FUNCTION_BLOCK "LOOP"   // FB2, LAD
{ S7_Optimized_Access := 'TRUE' }
VERSION : 0.1
// stored: AutoNumber true, IsIECCheckEnabled false, IsRetainMemResEnabled false, MemoryReserve 100, SetENOAutomatically false, UDAEnableTagReadback false
   VAR
      PULSO : Bool;
      AuxLoop : Bool;
      N_L00P : Int;
      Aux_N_LOOP : Int;
      Loop : Int;
   END_VAR
   VAR_TEMP   // added for the SCL form of the ladder/FBD networks
      _w1 : Bool;
      _w2 : Bool;
   END_VAR
BEGIN

REGION Network 2
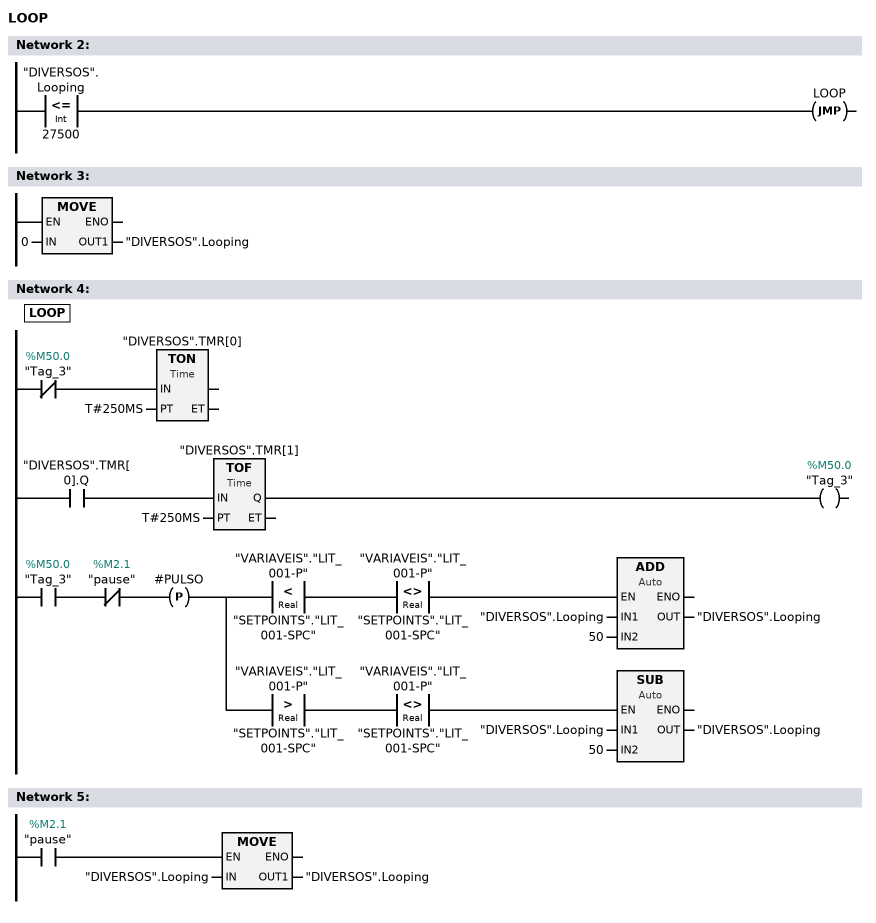
   RUNG wire#powerrail
      { S7_Templates := "SrcType := Int" } LE_Contact(in1 := "DIVERSOS".Looping, in2 := 27500)
      JumpCoil( LOOP )
   END_RUNG
   // the same network as SCL:
   IF "DIVERSOS".Looping <= 27500 THEN GOTO LOOP; END_IF;
END_REGION

REGION Network 3
   RUNG wire#powerrail
      Move(in := 0, out1 => "DIVERSOS".Looping)
   END_RUNG
   // the same network as SCL:
   "DIVERSOS".Looping := 0;
END_REGION

REGION Network 4
   Label( LOOP )
   RUNG wire#powerrail
      I_Contact( "Tag_3" )
      { S7_Templates := "time_type := Time" } "DIVERSOS".TMR[0].TON(pt := T#250MS, et =>)
   END_RUNG
   RUNG wire#powerrail
      Contact( "DIVERSOS".TMR[0].Q )
      { S7_Templates := "time_type := Time" } "DIVERSOS".TMR[1].TOF(pt := T#250MS, et =>)
      Coil( "Tag_3" )
   END_RUNG
   RUNG wire#powerrail
      Contact( "Tag_3" )
      I_Contact( "pause" )
      P_Trig( #PULSO )
      wire#w1
      { S7_Templates := "SrcType := Real" } LT_Contact(in1 := "VARIAVEIS"."LIT_001-P", in2 := "SETPOINTS"."LIT_001-SPC")
      { S7_Templates := "SrcType := Real" } NE_Contact(in1 := "VARIAVEIS"."LIT_001-P", in2 := "SETPOINTS"."LIT_001-SPC")
      Add(in1 := "DIVERSOS".Looping, in2 := 50, out => "DIVERSOS".Looping)
   END_RUNG
   RUNG wire#w1
      { S7_Templates := "SrcType := Real" } GT_Contact(in1 := "VARIAVEIS"."LIT_001-P", in2 := "SETPOINTS"."LIT_001-SPC")
      { S7_Templates := "SrcType := Real" } NE_Contact(in1 := "VARIAVEIS"."LIT_001-P", in2 := "SETPOINTS"."LIT_001-SPC")
      Sub(in1 := "DIVERSOS".Looping, in2 := 50, out => "DIVERSOS".Looping)
   END_RUNG
   // the same network as SCL:
   LOOP:
   "DIVERSOS".TMR[0].TON(IN := NOT "Tag_3", PT := T#250MS);
   "DIVERSOS".TMR[1].TOF(IN := "DIVERSOS".TMR[0].Q, PT := T#250MS);
   "Tag_3" := "DIVERSOS".TMR[1].Q;
   #_w1 := "Tag_3" AND NOT "pause";
   #_w2 := #_w1 AND NOT #PULSO;   // rising edge
   #PULSO := #_w1;
   IF #_w2 AND ("VARIAVEIS"."LIT_001-P" < "SETPOINTS"."LIT_001-SPC") AND ("VARIAVEIS"."LIT_001-P" <> "SETPOINTS"."LIT_001-SPC") THEN
       "DIVERSOS".Looping := "DIVERSOS".Looping + 50;
   END_IF;
   IF #_w2 AND ("VARIAVEIS"."LIT_001-P" > "SETPOINTS"."LIT_001-SPC") AND ("VARIAVEIS"."LIT_001-P" <> "SETPOINTS"."LIT_001-SPC") THEN
       "DIVERSOS".Looping := "DIVERSOS".Looping - 50;
   END_IF;
END_REGION

REGION Network 5
   RUNG wire#powerrail
      Contact( "pause" )
      Move(in := "DIVERSOS".Looping, out1 => "DIVERSOS".Looping)
   END_RUNG
   // the same network as SCL:
   IF "pause" THEN "DIVERSOS".Looping := "DIVERSOS".Looping; END_IF;
END_REGION
END_FUNCTION_BLOCK

FUNCTION_BLOCK "INTPRO"   // FB202, LAD
{ S7_Optimized_Access := 'FALSE' }
VERSION : 0.1
// stored: AutoNumber true, IsIECCheckEnabled false, SetENOAutomatically false, UDAEnableTagReadback false
   VAR DB_SPECIFIC
      EE_P_NIV : Bool;   // HAILITA BOMBA PRINCIPAL PELO NÍVEL
      EE_C1_NIV : Bool;   // HAILITA BOMBA COMPLEMENTAR 1 PELO NÍVEL
      EE_C2_NIV : Bool;   // HAILITA BOMBA COMPLEMENTAR 2 PELO NÍVEL
      EE_P_LS : Bool;   // HAILITA BOMBA PRINCIPAL PELAS BÓIAS
      EE_C1_LS : Bool;   // HAILITA BOMBA COMLEMENTAR 1 PELAS BÓIAS
      EE_C2_LS : Bool;   // HAILITA BOMBA COMPLEMENTAR 2 PELAS BÓIAS
      HAB_P_EE : Bool;   // LIGA BOMBA PRINCIPAL DA ELEVATÓRIA
      HAB_C1_EE : Bool;   // LIGA BOMBA COMPLEMENTAR 1 DA ELEVATÓRIA
      HAB_C2_EE : Bool;   // LIGA BOMBA COMPLEMENTAR 2 DA ELEVATÓRIA
      AUXP01 : Bool;
      BS01OK : Bool;
      BS02OK : Bool;
      BS03OK : Bool;
      L_BS01 : Bool;
      L_BS02 : Bool;
      L_BS03 : Bool;
      AUXP02 : Bool;
      AUXP03 : Bool;
      AUXP04 : Bool;
      AUXP05 : Bool;
      AUXP06 : Bool;
      AUXP07 : Bool;
      ETBS01_T001 : Int;
      ETBS02_T001 : Int;
      ETBS03_T001 : Int;
      BS01TO : Int;
      BS02TO : Int;
      BS03TO : Int;
      BS01TEOK : DInt;
      BS02TEOK : DInt;
      BS03TEOK : DInt;
      TE00 { S7_SetPoint := 'True'} : IEC_TIMER;
   END_VAR
   VAR
      RODEE { S7_SetPoint := 'True'} : "ROD4";
   END_VAR
   VAR_TEMP
      T011S : Int;
      ET_TE00 : Time;
   END_VAR
BEGIN

REGION Network 1: Alarme falha de sinal transmissor de nivel
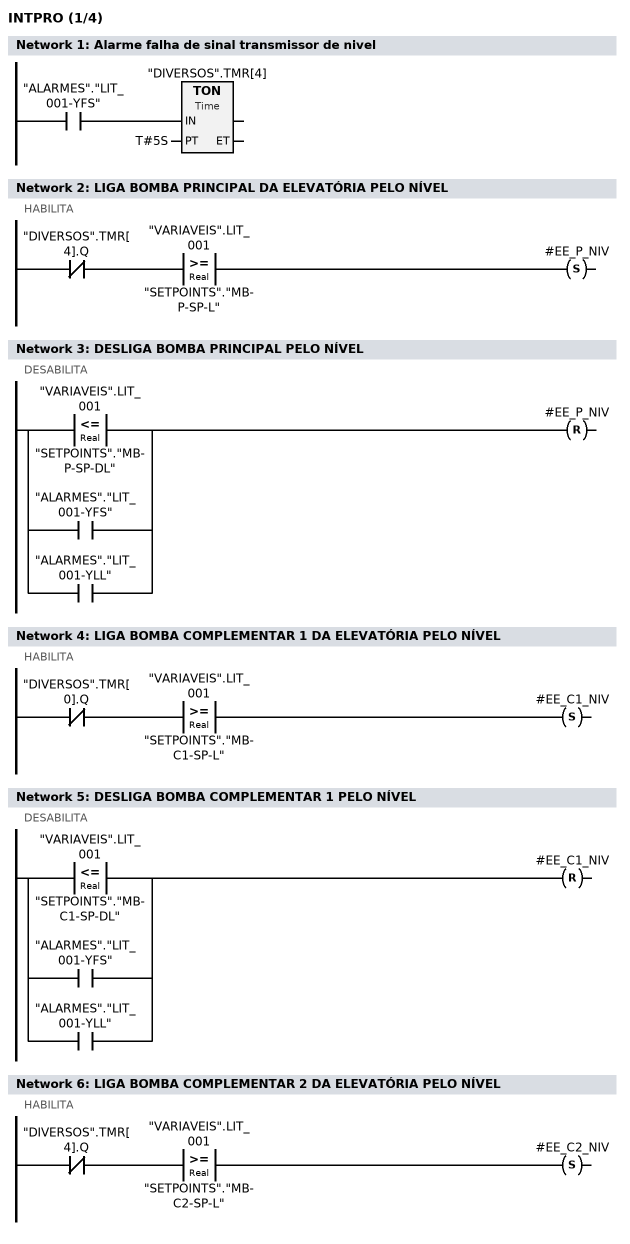
   RUNG wire#powerrail
      Contact( "ALARMES"."LIT_001-YFS" )
      { S7_Templates := "time_type := Time" } "DIVERSOS".TMR[4].TON(pt := T#5S, et =>)
   END_RUNG
   // the same network as SCL:
   "DIVERSOS".TMR[4].TON(IN := "ALARMES"."LIT_001-YFS", PT := T#5S);
END_REGION

REGION Network 2: LIGA BOMBA PRINCIPAL DA ELEVATÓRIA PELO NÍVEL
   // HABILITA
   RUNG wire#powerrail
      I_Contact( "DIVERSOS".TMR[4].Q )
      { S7_Templates := "SrcType := Real" } GE_Contact(in1 := "VARIAVEIS".LIT_001, in2 := "SETPOINTS"."MB-P-SP-L")
      S_Coil( #EE_P_NIV )
   END_RUNG
   // the same network as SCL:
   IF NOT "DIVERSOS".TMR[4].Q AND ("VARIAVEIS".LIT_001 >= "SETPOINTS"."MB-P-SP-L") THEN
       #EE_P_NIV := TRUE;
   END_IF;
END_REGION

REGION Network 3: DESLIGA BOMBA PRINCIPAL PELO NÍVEL
   // DESABILITA
   RUNG wire#powerrail
      { S7_Templates := "SrcType := Real" } LE_Contact(in1 := "VARIAVEIS".LIT_001, in2 := "SETPOINTS"."MB-P-SP-DL")
      wire#w1
      R_Coil( #EE_P_NIV )
   END_RUNG
   RUNG wire#powerrail
      Contact( "ALARMES"."LIT_001-YFS" )
   END_RUNG wire#w1
   RUNG wire#powerrail
      Contact( "ALARMES"."LIT_001-YLL" )
   END_RUNG wire#w1
   // the same network as SCL:
   IF ("VARIAVEIS".LIT_001 <= "SETPOINTS"."MB-P-SP-DL") OR "ALARMES"."LIT_001-YFS" OR "ALARMES"."LIT_001-YLL" THEN
       #EE_P_NIV := FALSE;
   END_IF;
END_REGION

REGION Network 4: LIGA BOMBA COMPLEMENTAR 1 DA ELEVATÓRIA PELO NÍVEL
   // HABILITA
   RUNG wire#powerrail
      I_Contact( "DIVERSOS".TMR[0].Q )
      { S7_Templates := "SrcType := Real" } GE_Contact(in1 := "VARIAVEIS".LIT_001, in2 := "SETPOINTS"."MB-C1-SP-L")
      S_Coil( #EE_C1_NIV )
   END_RUNG
   // the same network as SCL:
   IF NOT "DIVERSOS".TMR[0].Q AND ("VARIAVEIS".LIT_001 >= "SETPOINTS"."MB-C1-SP-L") THEN
       #EE_C1_NIV := TRUE;
   END_IF;
END_REGION

REGION Network 5: DESLIGA BOMBA COMPLEMENTAR 1 PELO NÍVEL
   // DESABILITA
   RUNG wire#powerrail
      { S7_Templates := "SrcType := Real" } LE_Contact(in1 := "VARIAVEIS".LIT_001, in2 := "SETPOINTS"."MB-C1-SP-DL")
      wire#w1
      R_Coil( #EE_C1_NIV )
   END_RUNG
   RUNG wire#powerrail
      Contact( "ALARMES"."LIT_001-YFS" )
   END_RUNG wire#w1
   RUNG wire#powerrail
      Contact( "ALARMES"."LIT_001-YLL" )
   END_RUNG wire#w1
   // the same network as SCL:
   IF ("VARIAVEIS".LIT_001 <= "SETPOINTS"."MB-C1-SP-DL") OR "ALARMES"."LIT_001-YFS" OR "ALARMES"."LIT_001-YLL" THEN
       #EE_C1_NIV := FALSE;
   END_IF;
END_REGION

REGION Network 6: LIGA BOMBA COMPLEMENTAR 2 DA ELEVATÓRIA PELO NÍVEL
   // HABILITA
   RUNG wire#powerrail
      I_Contact( "DIVERSOS".TMR[4].Q )
      { S7_Templates := "SrcType := Real" } GE_Contact(in1 := "VARIAVEIS".LIT_001, in2 := "SETPOINTS"."MB-C2-SP-L")
      S_Coil( #EE_C2_NIV )
   END_RUNG
   // the same network as SCL:
   IF NOT "DIVERSOS".TMR[4].Q AND ("VARIAVEIS".LIT_001 >= "SETPOINTS"."MB-C2-SP-L") THEN
       #EE_C2_NIV := TRUE;
   END_IF;
END_REGION

REGION Network 7: DESLIGA BOMBA COMPLEMENTAR 2 PELO NÍVEL
   // DESABILITA
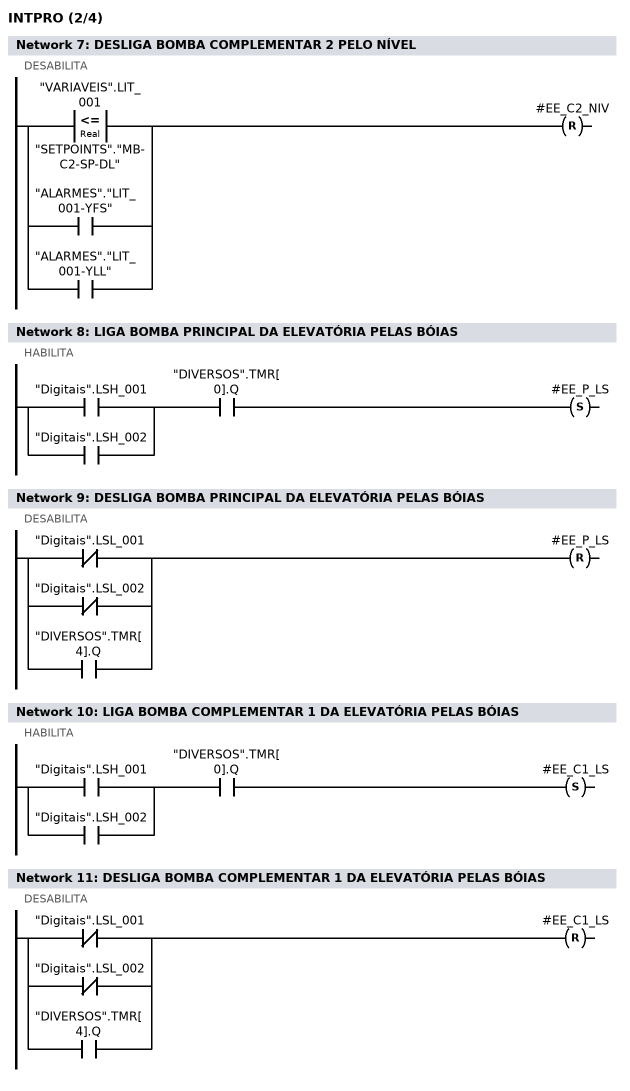
   RUNG wire#powerrail
      { S7_Templates := "SrcType := Real" } LE_Contact(in1 := "VARIAVEIS".LIT_001, in2 := "SETPOINTS"."MB-C2-SP-DL")
      wire#w1
      R_Coil( #EE_C2_NIV )
   END_RUNG
   RUNG wire#powerrail
      Contact( "ALARMES"."LIT_001-YFS" )
   END_RUNG wire#w1
   RUNG wire#powerrail
      Contact( "ALARMES"."LIT_001-YLL" )
   END_RUNG wire#w1
   // the same network as SCL:
   IF ("VARIAVEIS".LIT_001 <= "SETPOINTS"."MB-C2-SP-DL") OR "ALARMES"."LIT_001-YFS" OR "ALARMES"."LIT_001-YLL" THEN
       #EE_C2_NIV := FALSE;
   END_IF;
END_REGION

REGION Network 8: LIGA BOMBA PRINCIPAL DA ELEVATÓRIA PELAS BÓIAS
   // HABILITA
   RUNG wire#powerrail
      Contact( "Digitais".LSH_001 )
      wire#w1
      Contact( "DIVERSOS".TMR[0].Q )
      S_Coil( #EE_P_LS )
   END_RUNG
   RUNG wire#powerrail
      Contact( "Digitais".LSH_002 )
   END_RUNG wire#w1
   // the same network as SCL:
   IF ("Digitais".LSH_001 OR "Digitais".LSH_002) AND "DIVERSOS".TMR[0].Q THEN #EE_P_LS := TRUE; END_IF;
END_REGION

REGION Network 9: DESLIGA BOMBA PRINCIPAL DA ELEVATÓRIA PELAS BÓIAS
   // DESABILITA
   RUNG wire#powerrail
      I_Contact( "Digitais".LSL_001 )
      wire#w1
      R_Coil( #EE_P_LS )
   END_RUNG
   RUNG wire#powerrail
      I_Contact( "Digitais".LSL_002 )
   END_RUNG wire#w1
   RUNG wire#powerrail
      Contact( "DIVERSOS".TMR[4].Q )
   END_RUNG wire#w1
   // the same network as SCL:
   IF NOT "Digitais".LSL_001 OR NOT "Digitais".LSL_002 OR "DIVERSOS".TMR[4].Q THEN #EE_P_LS := FALSE; END_IF;
END_REGION

REGION Network 10: LIGA BOMBA COMPLEMENTAR 1 DA ELEVATÓRIA PELAS BÓIAS
   // HABILITA
   RUNG wire#powerrail
      Contact( "Digitais".LSH_001 )
      wire#w1
      Contact( "DIVERSOS".TMR[0].Q )
      S_Coil( #EE_C1_LS )
   END_RUNG
   RUNG wire#powerrail
      Contact( "Digitais".LSH_002 )
   END_RUNG wire#w1
   // the same network as SCL:
   IF ("Digitais".LSH_001 OR "Digitais".LSH_002) AND "DIVERSOS".TMR[0].Q THEN #EE_C1_LS := TRUE; END_IF;
END_REGION

REGION Network 11: DESLIGA BOMBA COMPLEMENTAR 1 DA ELEVATÓRIA PELAS BÓIAS
   // DESABILITA
   RUNG wire#powerrail
      I_Contact( "Digitais".LSL_001 )
      wire#w1
      R_Coil( #EE_C1_LS )
   END_RUNG
   RUNG wire#powerrail
      I_Contact( "Digitais".LSL_002 )
   END_RUNG wire#w1
   RUNG wire#powerrail
      Contact( "DIVERSOS".TMR[4].Q )
   END_RUNG wire#w1
   // the same network as SCL:
   IF NOT "Digitais".LSL_001 OR NOT "Digitais".LSL_002 OR "DIVERSOS".TMR[4].Q THEN
       #EE_C1_LS := FALSE;
   END_IF;
END_REGION

REGION Network 12: LIGA BOMBA COMPLEMENTAR 2 DA ELEVATÓRIA PELAS BÓIAS
   // HABILITA
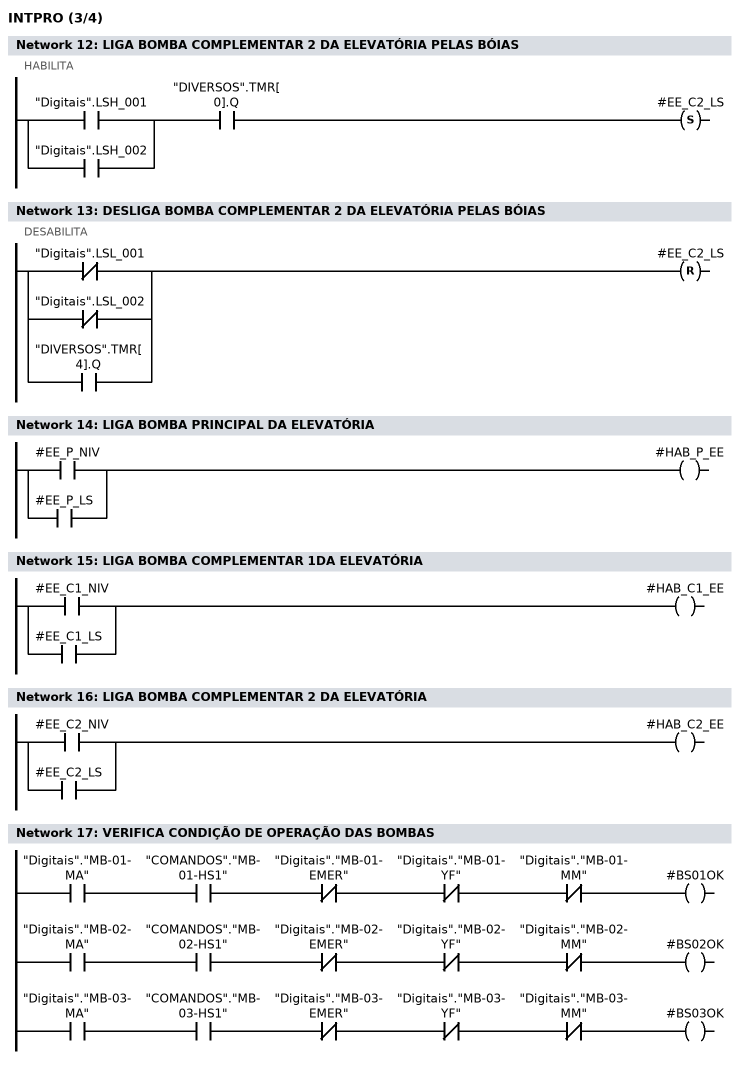
   RUNG wire#powerrail
      Contact( "Digitais".LSH_001 )
      wire#w1
      Contact( "DIVERSOS".TMR[0].Q )
      S_Coil( #EE_C2_LS )
   END_RUNG
   RUNG wire#powerrail
      Contact( "Digitais".LSH_002 )
   END_RUNG wire#w1
   // the same network as SCL:
   IF ("Digitais".LSH_001 OR "Digitais".LSH_002) AND "DIVERSOS".TMR[0].Q THEN #EE_C2_LS := TRUE; END_IF;
END_REGION

REGION Network 13: DESLIGA BOMBA COMPLEMENTAR 2 DA ELEVATÓRIA PELAS BÓIAS
   // DESABILITA
   RUNG wire#powerrail
      I_Contact( "Digitais".LSL_001 )
      wire#w1
      R_Coil( #EE_C2_LS )
   END_RUNG
   RUNG wire#powerrail
      I_Contact( "Digitais".LSL_002 )
   END_RUNG wire#w1
   RUNG wire#powerrail
      Contact( "DIVERSOS".TMR[4].Q )
   END_RUNG wire#w1
   // the same network as SCL:
   IF NOT "Digitais".LSL_001 OR NOT "Digitais".LSL_002 OR "DIVERSOS".TMR[4].Q THEN
       #EE_C2_LS := FALSE;
   END_IF;
END_REGION

REGION Network 14: LIGA BOMBA PRINCIPAL DA ELEVATÓRIA
   RUNG wire#powerrail
      Contact( #EE_P_NIV )
      wire#w1
      Coil( #HAB_P_EE )
   END_RUNG
   RUNG wire#powerrail
      Contact( #EE_P_LS )
   END_RUNG wire#w1
   // the same network as SCL:
   #HAB_P_EE := #EE_P_NIV OR #EE_P_LS;
END_REGION

REGION Network 15: LIGA BOMBA COMPLEMENTAR 1DA ELEVATÓRIA
   RUNG wire#powerrail
      Contact( #EE_C1_NIV )
      wire#w1
      Coil( #HAB_C1_EE )
   END_RUNG
   RUNG wire#powerrail
      Contact( #EE_C1_LS )
   END_RUNG wire#w1
   // the same network as SCL:
   #HAB_C1_EE := #EE_C1_NIV OR #EE_C1_LS;
END_REGION

REGION Network 16: LIGA BOMBA COMPLEMENTAR 2 DA ELEVATÓRIA
   RUNG wire#powerrail
      Contact( #EE_C2_NIV )
      wire#w1
      Coil( #HAB_C2_EE )
   END_RUNG
   RUNG wire#powerrail
      Contact( #EE_C2_LS )
   END_RUNG wire#w1
   // the same network as SCL:
   #HAB_C2_EE := #EE_C2_NIV OR #EE_C2_LS;
END_REGION

REGION Network 17: VERIFICA CONDIÇÃO DE OPERAÇÃO DAS BOMBAS
   RUNG wire#powerrail
      Contact( "Digitais"."MB-01-MA" )
      Contact( "COMANDOS"."MB-01-HS1" )
      I_Contact( "Digitais"."MB-01-EMER" )
      I_Contact( "Digitais"."MB-01-YF" )
      I_Contact( "Digitais"."MB-01-MM" )
      Coil( #BS01OK )
   END_RUNG
   RUNG wire#powerrail
      Contact( "Digitais"."MB-02-MA" )
      Contact( "COMANDOS"."MB-02-HS1" )
      I_Contact( "Digitais"."MB-02-EMER" )
      I_Contact( "Digitais"."MB-02-YF" )
      I_Contact( "Digitais"."MB-02-MM" )
      Coil( #BS02OK )
   END_RUNG
   RUNG wire#powerrail
      Contact( "Digitais"."MB-03-MA" )
      Contact( "COMANDOS"."MB-03-HS1" )
      I_Contact( "Digitais"."MB-03-EMER" )
      I_Contact( "Digitais"."MB-03-YF" )
      I_Contact( "Digitais"."MB-03-MM" )
      Coil( #BS03OK )
   END_RUNG
   // the same network as SCL:
   #BS01OK := "Digitais"."MB-01-MA" AND "COMANDOS"."MB-01-HS1" AND NOT "Digitais"."MB-01-EMER" AND NOT "Digitais"."MB-01-YF" AND NOT "Digitais"."MB-01-MM";
   #BS02OK := "Digitais"."MB-02-MA" AND "COMANDOS"."MB-02-HS1" AND NOT "Digitais"."MB-02-EMER" AND NOT "Digitais"."MB-02-YF" AND NOT "Digitais"."MB-02-MM";
   #BS03OK := "Digitais"."MB-03-MA" AND "COMANDOS"."MB-03-HS1" AND NOT "Digitais"."MB-03-EMER" AND NOT "Digitais"."MB-03-YF" AND NOT "Digitais"."MB-03-MM";
END_REGION

REGION Network 18: RODÍZIO DAS BOMBAS
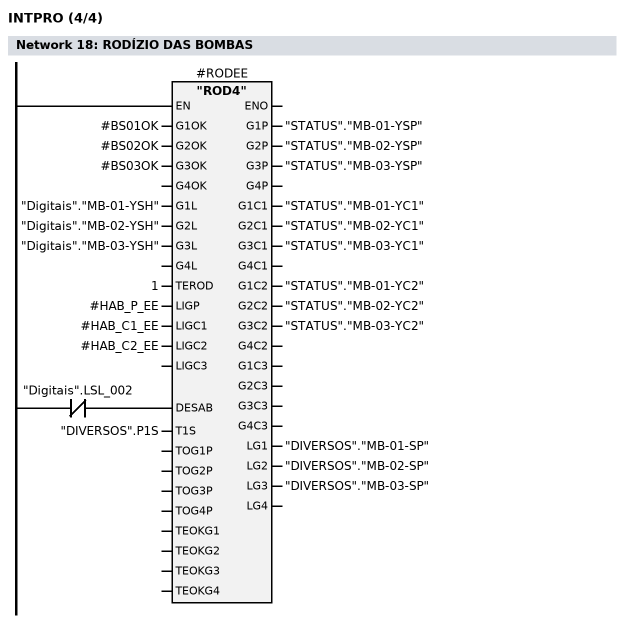
   RUNG wire#powerrail
      #RODEE(DESAB := wire#w1, G1OK := #BS01OK, G2OK := #BS02OK, G3OK := #BS03OK, G4OK :=, G1L := "Digitais"."MB-01-YSH", G2L := "Digitais"."MB-02-YSH", G3L := "Digitais"."MB-03-YSH", G4L :=, TEROD := 1, LIGP := #HAB_P_EE, LIGC1 := #HAB_C1_EE, LIGC2 := #HAB_C2_EE, LIGC3 :=, T1S := "DIVERSOS".P1S, TOG1P :=, TOG2P :=, TOG3P :=, TOG4P :=, TEOKG1 :=, TEOKG2 :=, TEOKG3 :=, TEOKG4 :=, G1P => "STATUS"."MB-01-YSP", G2P => "STATUS"."MB-02-YSP", G3P => "STATUS"."MB-03-YSP", G4P =>, G1C1 => "STATUS"."MB-01-YC1", G2C1 => "STATUS"."MB-02-YC1", G3C1 => "STATUS"."MB-03-YC1", G4C1 =>, G1C2 => "STATUS"."MB-01-YC2", G2C2 => "STATUS"."MB-02-YC2", G3C2 => "STATUS"."MB-03-YC2", G4C2 =>, G1C3 =>, G2C3 =>, G3C3 =>, G4C3 =>, LG1 => "DIVERSOS"."MB-01-SP", LG2 => "DIVERSOS"."MB-02-SP", LG3 => "DIVERSOS"."MB-03-SP", LG4 =>)
   END_RUNG
   RUNG wire#powerrail
      I_Contact( "Digitais".LSL_002 )
   END_RUNG wire#w1
   // the same network as SCL:
   #RODEE(G1OK := #BS01OK,   // "ROD4"
          G2OK := #BS02OK,
          G3OK := #BS03OK,
          G1L := "Digitais"."MB-01-YSH",
          G2L := "Digitais"."MB-02-YSH",
          G3L := "Digitais"."MB-03-YSH",
          TEROD := 1,
          LIGP := #HAB_P_EE,
          LIGC1 := #HAB_C1_EE,
          LIGC2 := #HAB_C2_EE,
          DESAB := NOT "Digitais".LSL_002,
          T1S := "DIVERSOS".P1S,
          G1P => "STATUS"."MB-01-YSP",
          G2P => "STATUS"."MB-02-YSP",
          G3P => "STATUS"."MB-03-YSP",
          G1C1 => "STATUS"."MB-01-YC1",
          G2C1 => "STATUS"."MB-02-YC1",
          G3C1 => "STATUS"."MB-03-YC1",
          G1C2 => "STATUS"."MB-01-YC2",
          G2C2 => "STATUS"."MB-02-YC2",
          G3C2 => "STATUS"."MB-03-YC2",
          LG1 => "DIVERSOS"."MB-01-SP",
          LG2 => "DIVERSOS"."MB-02-SP",
          LG3 => "DIVERSOS"."MB-03-SP");
END_REGION
END_FUNCTION_BLOCK

FUNCTION_BLOCK "ROD4"   // FB200, LAD
TITLE = Rodízio de 4 grupos
{ S7_Optimized_Access := 'FALSE' }
VERSION : 0.1
// stored: AutoNumber false, IsIECCheckEnabled false, SetENOAutomatically false, UDAEnableTagReadback false
   VAR_INPUT
      G1OK : Bool;   // GRUPO EM CONDIÇÕES DE OPERAÇÃO
      G2OK : Bool;   // GRUPO EM CONDIÇÕES DE OPERAÇÃO
      G3OK : Bool;   // GRUPO EM CONDIÇÕES DE OPERAÇÃO
      G4OK : Bool;   // GRUPO EM CONDIÇÕES DE OPERAÇÃO
      G1L : Bool;   // GRUPO LIGADO
      G2L : Bool;   // GRUPO LIGADO
      G3L : Bool;   // GRUPO LIGADO
      G4L : Bool;   // GRUPO LIGADO
      TEROD : DInt;   // TEMPOPARA RODÍZIO DAS BOMBAS
      LIGP : Bool;   // LIGA BOMBA PRINCIPAL
      LIGC1 : Bool;   // LIGA BOMBA COMPLEMENTAR 1
      LIGC2 : Bool;   // LIGA BOMBA COMPLEMENTAR 2
      LIGC3 : Bool;   // LIGA BOMBA COMPLEMENTAR 3
      DESAB : Bool;   // DESABILITA FUNCIONAMENTO DOS GRUPOS
      T1S : Bool;   // PULSO A CADA 1 SEGUNDO
   END_VAR
   VAR_OUTPUT
      G1P : Bool;   // GRUPO 1 SELECIONADO COMO PRINCIPAL
      G2P : Bool;   // GRUPO 2 SELECIONADO COMO PRINCIPAL
      G3P : Bool;   // GRUPO 3 SELECIONADO COMO PRINCIPAL
      G4P : Bool;   // GRUPO 4 SELECIONADO COMO PRINCIPAL
      G1C1 : Bool;   // GRUPO 1 SELECIONADO COMO COMPLEMENTAR 1
      G2C1 : Bool;   // GRUPO 2 SELECIONADO COMO COMPLEMENTAR 1
      G3C1 : Bool;   // GRUPO 3 SELECIONADO COMO COMPLEMENTAR 1
      G4C1 : Bool;   // GRUPO 4 SELECIONADO COMO COMPLEMENTAR 1
      G1C2 : Bool;   // GRUPO 1 SELECIONADO COMO COMPLEMENTAR 2
      G2C2 : Bool;   // GRUPO 2 SELECIONADO COMO COMPLEMENTAR 2
      G3C2 : Bool;   // GRUPO 3 SELECIONADO COMO COMPLEMENTAR 3
      G4C2 : Bool;   // GRUPO 4 SELECIONADO COMO COMPLEMENTAR 4
      G1C3 : Bool;   // GRUPO 1 SELECIONADO COMO COMPLEMENTAR 3
      G2C3 : Bool;   // GRUPO 2 SELECIONADO COMO COMPLEMENTAR 3
      G3C3 : Bool;   // GRUPO 3 SELECIONADO COMO COMPLEMENTAR 3
      G4C3 : Bool;   // GRUPO 4 SELECIONADO COMO COMPLEMENTAR 3
      LG1 : Bool;   // LIGA GRUPO 1
      LG2 : Bool;   // LIGA GRUPO 2
      LG3 : Bool;   // LIGA GRUPO 3
      LG4 : Bool;   // LIGA GRUPO 4
   END_VAR
   VAR_IN_OUT
      TOG1P : DInt;   // TEMPO DE OPERAÇÃO GRUPO 1
      TOG2P : DInt;   // TEMPO DE OPERAÇÃO GRUPO 2
      TOG3P : DInt;   // TEMPO DE OPERAÇÃO GRUPO 3
      TOG4P : DInt;   // TEMPO DE OPERAÇÃO GRUPO 4
      TEOKG1 : Real;   // TEMPO OK GRUPO 1
      TEOKG2 : Real;   // TEMPO OK GRUPO 2
      TEOKG3 : Real;   // TEMPO OK GRUPO 3
      TEOKG4 : Real;   // TEMPO OK GRUPO 4
   END_VAR
   VAR DB_SPECIFIC
      GR1SELP : Bool;   // SELECIONADO COMO PRINCIPAL
      GR2SELP : Bool;   // SELECIONADO COMO PRINCIPAL
      GR3SELP : Bool;   // SELECIONADO COMO PRINCIPAL
      GR4SELP : Bool;   // SELECIONADO COMO PRINCIPAL
      GR1SELC1 : Bool;   // SELECIONADO COMO COMPLEMENTAR 1
      GR2SELC1 : Bool;   // SELECIONADO COMO COMPLEMENTAR 1
      GR3SELC1 : Bool;   // SELECIONADO COMO COMPLEMENTAR 1
      GR4SELC1 : Bool;   // SELECIONADO COMO COMPLEMENTAR 1
      GR1SELC2 : Bool;   // SELECIONADO COMO COMPLEMENTAR 2
      GR2SELC2 : Bool;   // SELECIONADO COMO COMPLEMENTAR 2
      GR3SELC2 : Bool;   // SELECIONADO COMO COMPLEMENTAR 2
      GR4SELC2 : Bool;   // SELECIONADO COMO COMPLEMENTAR 2
      GR1SELC3 : Bool;   // SELECIONADO COMO COMPLEMENTAR 3
      GR2SELC3 : Bool;   // SELECIONADO COMO COMPLEMENTAR 3
      GR3SELC3 : Bool;   // SELECIONADO COMO COMPLEMENTAR 3
      GR4SELC3 : Bool;   // SELECIONADO COMO COMPLEMENTAR 3
      PS1SG1 : Bool;   // AUXILIAR DE PULSO
      PS1SG2 : Bool;   // AUXILIAR DE PULSO
      PS1SG3 : Bool;   // AUXILIAR DE PULSO
      PS1SG4 : Bool;   // AUXILIAR DE PULSO
      PS1 : Bool;   // AUXILIAR DE PULSO
      PS2 : Bool;   // AUXILIAR DE PULSO
      PS3 : Bool;   // AUXILIAR DE PULSO
      PS4 : Bool;   // AUXILIAR DE PULSO
      FIMTEG1 : Bool;   // FIM DO TEMPO DE EXISTÊNCIA DO GRUPO 1
      FIMTEG2 : Bool;   // FIM DO TEMPO DE EXISTÊNCIA DO GRUPO 2
      FIMTEG3 : Bool;   // FIM DO TEMPO DE EXISTÊNCIA DO GRUPO 3
      FIMTEG4 : Bool;   // FIM DO TEMPO DE EXISTÊNCIA DO GRUPO 4
      SDESG1 : Bool;   // SOLICITAÇÃO DE DESLIGAMENTO
      SDESG2 : Bool;   // SOLICITAÇÃO DE DESLIGAMENTO
      SDESG3 : Bool;   // SOLICITAÇÃO DE DESLIGAMENTO
      SDESG4 : Bool;   // SOLICITAÇÃO DE DESLIGAMENTO
      GPL : Bool;   // GRUPO PRINCIPAL LIGADO
      GC1L : Bool;   // GRUPO COMPLEMENTAR 1 LIGADO
      GC2L : Bool;   // GRUPO COMPLEMENTAR 2 LIGADO
      GC3L : Bool;   // GRUPO COMPLEMENTAR 3 LIGADO
      SO_L : Bool;   // SOLICITAÇÃO DE PARTIDA
      SO_D : Bool;   // SOLICITAÇÃO DE DESLIGAMENTO
      RTEOKG1 : Bool;   // RESET TEMPO OK
      RTEOKG2 : Bool;   // RESET TEMPO OK
      RTEOKG3 : Bool;   // RESET TEMPO OK
      RTEOKG4 : Bool;   // RESET TEMPO OK
      TON1 { S7_SetPoint := 'True'} : TON_TIME;   // TEMPORIZADOR
      TON2 { S7_SetPoint := 'True'} : TON_TIME;   // TEMPORIZADOR
      TON3 { S7_SetPoint := 'True'} : TON_TIME;   // TEMPORIZADOR
      TON4 { S7_SetPoint := 'True'} : TON_TIME;   // TEMPORIZADOR
      TSDG1 { S7_SetPoint := 'True'} : TON_TIME;   // TEMPORIZADOR
      TSDG2 { S7_SetPoint := 'True'} : TON_TIME;   // TEMPORIZADOR
      TSDG3 { S7_SetPoint := 'True'} : TON_TIME;   // TEMPORIZADOR
      TSDG4 { S7_SetPoint := 'True'} : TON_TIME;   // TEMPORIZADOR
   END_VAR
   VAR_TEMP
      PRI12 : Bool;   // PRIORIDADE GRUPO 1
      PRI13 : Bool;   // PRIORIDADE GRUPO 1
      PRI14 : Bool;   // PRIORIDADE GRUPO 1
      PRI23 : Bool;   // PRIORIDADE GRUPO 2
      PRI24 : Bool;   // PRIORIDADE GRUPO 2
      PRI34 : Bool;   // PRIORIDADE GRUPO 3
      TMROD : Real;   // TEMPO DE RODIZIO
      NGS : Int;   // NÚMERO DE GRUPOS SOLICITADOS
      NGF : Int;   // NÚMERO DE GRUPOS FUNCIONANDO
      AUX01 : Int;   // AUXILIAR UTILIZADO NA LÓGICA
      AUX02 : Int;   // AUXILIAR UTILIZADO NA LÓGICA
      AUX03 : Int;   // AUXILIAR UTILIZADO NA LÓGICA
      AUX04 : Int;   // AUXILIAR UTILIZADO NA LÓGICA
      AUX05 : Bool;   // AUXILIAR UTILIZADO NA LÓGICA
      AUX06 : Bool;   // AUXILIAR UTILIZADO NA LÓGICA
      AUX07 : Bool;   // AUXILIAR UTILIZADO NA LÓGICA
      AUX08 : Bool;   // AUXILIAR UTILIZADO NA LÓGICA
      ETT1 : Time;   // EFETIVO DO TEMPORIZADOR
      ETT2 : Time;   // EFETIVO DO TEMPORIZADOR
      ETT3 : Time;   // EFETIVO DO TEMPORIZADOR
      ETT4 : Time;   // EFETIVO DO TEMPORIZADOR
      ETTSDG4 : Time;   // EFETIVO DO TEMPORIZADOR
      ETTSDG3 : Time;   // EFETIVO DO TEMPORIZADOR
      ETTSDG2 : Time;   // EFETIVO DO TEMPORIZADOR
      ETTSDG1 : Time;   // EFETIVO DO TEMPORIZADOR
   END_VAR
   VAR_TEMP   // added for the SCL form of the ladder/FBD networks
      _w1 : Bool;
   END_VAR
BEGIN

REGION Network 1: Tranforme em segundo o tempo de rodízio dos sopradores
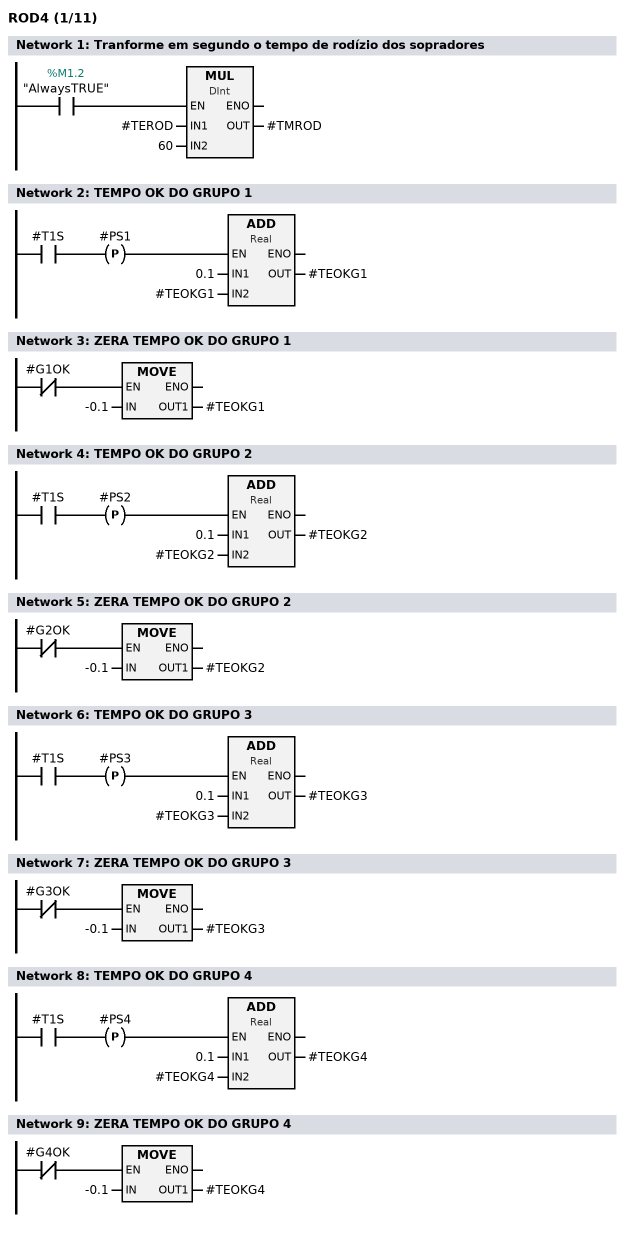
   RUNG wire#powerrail
      Contact( "AlwaysTRUE" )
      { S7_Templates := "SrcType := DInt"; S7_GenerateENO := "TRUE" } Mul(in1 := #TEROD, in2 := 60, out => #TMROD)
   END_RUNG
   // the same network as SCL:
   IF "AlwaysTRUE" THEN #TMROD := #TEROD * 60; END_IF;
END_REGION

REGION Network 2: TEMPO OK DO GRUPO 1
   RUNG wire#powerrail
      Contact( #T1S )
      P_Trig( #PS1 )
      { S7_Templates := "SrcType := Real"; S7_GenerateENO := "TRUE" } Add(in1 := 0.1, in2 := #TEOKG1, out => #TEOKG1)
   END_RUNG
   // the same network as SCL:
   #_w1 := #T1S AND NOT #PS1;   // rising edge
   #PS1 := #T1S;
   IF #_w1 THEN #TEOKG1 := 0.1 + #TEOKG1; END_IF;
END_REGION

REGION Network 3: ZERA TEMPO OK DO GRUPO 1
   RUNG wire#powerrail
      I_Contact( #G1OK )
      { S7_GenerateENO := "TRUE" } Move(in := -0.1, out1 => #TEOKG1)
   END_RUNG
   // the same network as SCL:
   IF NOT #G1OK THEN #TEOKG1 := -0.1; END_IF;
END_REGION

REGION Network 4: TEMPO OK DO GRUPO 2
   RUNG wire#powerrail
      Contact( #T1S )
      P_Trig( #PS2 )
      { S7_Templates := "SrcType := Real"; S7_GenerateENO := "TRUE" } Add(in1 := 0.1, in2 := #TEOKG2, out => #TEOKG2)
   END_RUNG
   // the same network as SCL:
   #_w1 := #T1S AND NOT #PS2;   // rising edge
   #PS2 := #T1S;
   IF #_w1 THEN #TEOKG2 := 0.1 + #TEOKG2; END_IF;
END_REGION

REGION Network 5: ZERA TEMPO OK DO GRUPO 2
   RUNG wire#powerrail
      I_Contact( #G2OK )
      { S7_GenerateENO := "TRUE" } Move(in := -0.1, out1 => #TEOKG2)
   END_RUNG
   // the same network as SCL:
   IF NOT #G2OK THEN #TEOKG2 := -0.1; END_IF;
END_REGION

REGION Network 6: TEMPO OK DO GRUPO 3
   RUNG wire#powerrail
      Contact( #T1S )
      P_Trig( #PS3 )
      { S7_Templates := "SrcType := Real"; S7_GenerateENO := "TRUE" } Add(in1 := 0.1, in2 := #TEOKG3, out => #TEOKG3)
   END_RUNG
   // the same network as SCL:
   #_w1 := #T1S AND NOT #PS3;   // rising edge
   #PS3 := #T1S;
   IF #_w1 THEN #TEOKG3 := 0.1 + #TEOKG3; END_IF;
END_REGION

REGION Network 7: ZERA TEMPO OK DO GRUPO 3
   RUNG wire#powerrail
      I_Contact( #G3OK )
      { S7_GenerateENO := "TRUE" } Move(in := -0.1, out1 => #TEOKG3)
   END_RUNG
   // the same network as SCL:
   IF NOT #G3OK THEN #TEOKG3 := -0.1; END_IF;
END_REGION

REGION Network 8: TEMPO OK DO GRUPO 4
   RUNG wire#powerrail
      Contact( #T1S )
      P_Trig( #PS4 )
      { S7_Templates := "SrcType := Real"; S7_GenerateENO := "TRUE" } Add(in1 := 0.1, in2 := #TEOKG4, out => #TEOKG4)
   END_RUNG
   // the same network as SCL:
   #_w1 := #T1S AND NOT #PS4;   // rising edge
   #PS4 := #T1S;
   IF #_w1 THEN #TEOKG4 := 0.1 + #TEOKG4; END_IF;
END_REGION

REGION Network 9: ZERA TEMPO OK DO GRUPO 4
   RUNG wire#powerrail
      I_Contact( #G4OK )
      { S7_GenerateENO := "TRUE" } Move(in := -0.1, out1 => #TEOKG4)
   END_RUNG
   // the same network as SCL:
   IF NOT #G4OK THEN #TEOKG4 := -0.1; END_IF;
END_REGION

REGION Network 10: DEFINIÇÇÃO DE PRIORIDADE DO GRUPO 1
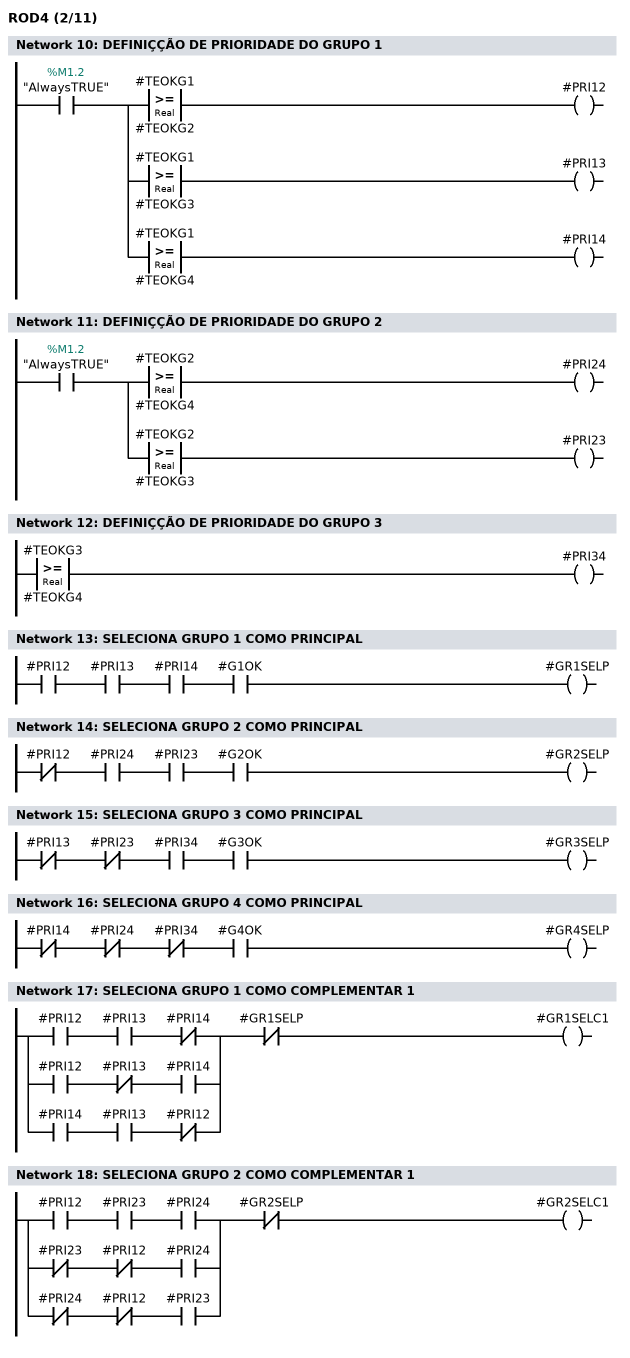
   RUNG wire#powerrail
      Contact( "AlwaysTRUE" )
      wire#w1
      { S7_Templates := "SrcType := Real" } GE_Contact(in1 := #TEOKG1, in2 := #TEOKG2)
      Coil( #PRI12 )
   END_RUNG
   RUNG wire#w1
      { S7_Templates := "SrcType := Real" } GE_Contact(in1 := #TEOKG1, in2 := #TEOKG3)
      Coil( #PRI13 )
   END_RUNG
   RUNG wire#w1
      { S7_Templates := "SrcType := Real" } GE_Contact(in1 := #TEOKG1, in2 := #TEOKG4)
      Coil( #PRI14 )
   END_RUNG
   // the same network as SCL:
   #PRI12 := "AlwaysTRUE" AND (#TEOKG1 >= #TEOKG2);
   #PRI13 := "AlwaysTRUE" AND (#TEOKG1 >= #TEOKG3);
   #PRI14 := "AlwaysTRUE" AND (#TEOKG1 >= #TEOKG4);
END_REGION

REGION Network 11: DEFINIÇÇÃO DE PRIORIDADE DO GRUPO 2
   RUNG wire#powerrail
      Contact( "AlwaysTRUE" )
      wire#w1
      { S7_Templates := "SrcType := Real" } GE_Contact(in1 := #TEOKG2, in2 := #TEOKG4)
      Coil( #PRI24 )
   END_RUNG
   RUNG wire#w1
      { S7_Templates := "SrcType := Real" } GE_Contact(in1 := #TEOKG2, in2 := #TEOKG3)
      Coil( #PRI23 )
   END_RUNG
   // the same network as SCL:
   #PRI24 := "AlwaysTRUE" AND (#TEOKG2 >= #TEOKG4);
   #PRI23 := "AlwaysTRUE" AND (#TEOKG2 >= #TEOKG3);
END_REGION

REGION Network 12: DEFINIÇÇÃO DE PRIORIDADE DO GRUPO 3
   RUNG wire#powerrail
      { S7_Templates := "SrcType := Real" } GE_Contact(in1 := #TEOKG3, in2 := #TEOKG4)
      Coil( #PRI34 )
   END_RUNG
   // the same network as SCL:
   #PRI34 := #TEOKG3 >= #TEOKG4;
END_REGION

REGION Network 13: SELECIONA GRUPO 1 COMO PRINCIPAL
   RUNG wire#powerrail
      Contact( #PRI12 )
      Contact( #PRI13 )
      Contact( #PRI14 )
      Contact( #G1OK )
      Coil( #GR1SELP )
   END_RUNG
   // the same network as SCL:
   #GR1SELP := #PRI12 AND #PRI13 AND #PRI14 AND #G1OK;
END_REGION

REGION Network 14: SELECIONA GRUPO 2 COMO PRINCIPAL
   RUNG wire#powerrail
      I_Contact( #PRI12 )
      Contact( #PRI24 )
      Contact( #PRI23 )
      Contact( #G2OK )
      Coil( #GR2SELP )
   END_RUNG
   // the same network as SCL:
   #GR2SELP := NOT #PRI12 AND #PRI24 AND #PRI23 AND #G2OK;
END_REGION

REGION Network 15: SELECIONA GRUPO 3 COMO PRINCIPAL
   RUNG wire#powerrail
      I_Contact( #PRI13 )
      I_Contact( #PRI23 )
      Contact( #PRI34 )
      Contact( #G3OK )
      Coil( #GR3SELP )
   END_RUNG
   // the same network as SCL:
   #GR3SELP := NOT #PRI13 AND NOT #PRI23 AND #PRI34 AND #G3OK;
END_REGION

REGION Network 16: SELECIONA GRUPO 4 COMO PRINCIPAL
   RUNG wire#powerrail
      I_Contact( #PRI14 )
      I_Contact( #PRI24 )
      I_Contact( #PRI34 )
      Contact( #G4OK )
      Coil( #GR4SELP )
   END_RUNG
   // the same network as SCL:
   #GR4SELP := NOT #PRI14 AND NOT #PRI24 AND NOT #PRI34 AND #G4OK;
END_REGION

REGION Network 17: SELECIONA GRUPO 1 COMO COMPLEMENTAR 1
   RUNG wire#powerrail
      Contact( #PRI12 )
      Contact( #PRI13 )
      I_Contact( #PRI14 )
      wire#w1
      I_Contact( #GR1SELP )
      Coil( #GR1SELC1 )
   END_RUNG
   RUNG wire#powerrail
      Contact( #PRI12 )
      I_Contact( #PRI13 )
      Contact( #PRI14 )
   END_RUNG wire#w1
   RUNG wire#powerrail
      Contact( #PRI14 )
      Contact( #PRI13 )
      I_Contact( #PRI12 )
   END_RUNG wire#w1
   // the same network as SCL:
   #GR1SELC1 := ((#PRI12 AND #PRI13 AND NOT #PRI14) OR (#PRI12 AND NOT #PRI13 AND #PRI14) OR (#PRI14 AND #PRI13 AND NOT #PRI12)) AND NOT #GR1SELP;
END_REGION

REGION Network 18: SELECIONA GRUPO 2 COMO COMPLEMENTAR 1
   RUNG wire#powerrail
      Contact( #PRI12 )
      Contact( #PRI23 )
      Contact( #PRI24 )
      wire#w1
      I_Contact( #GR2SELP )
      Coil( #GR2SELC1 )
   END_RUNG
   RUNG wire#powerrail
      I_Contact( #PRI23 )
      I_Contact( #PRI12 )
      Contact( #PRI24 )
   END_RUNG wire#w1
   RUNG wire#powerrail
      I_Contact( #PRI24 )
      I_Contact( #PRI12 )
      Contact( #PRI23 )
   END_RUNG wire#w1
   // the same network as SCL:
   #GR2SELC1 := ((#PRI12 AND #PRI23 AND #PRI24) OR (NOT #PRI23 AND NOT #PRI12 AND #PRI24) OR (NOT #PRI24 AND NOT #PRI12 AND #PRI23)) AND NOT #GR2SELP;
END_REGION

REGION Network 19: SELECIONA GRUPO 3 COMO COMPLEMENTAR 1
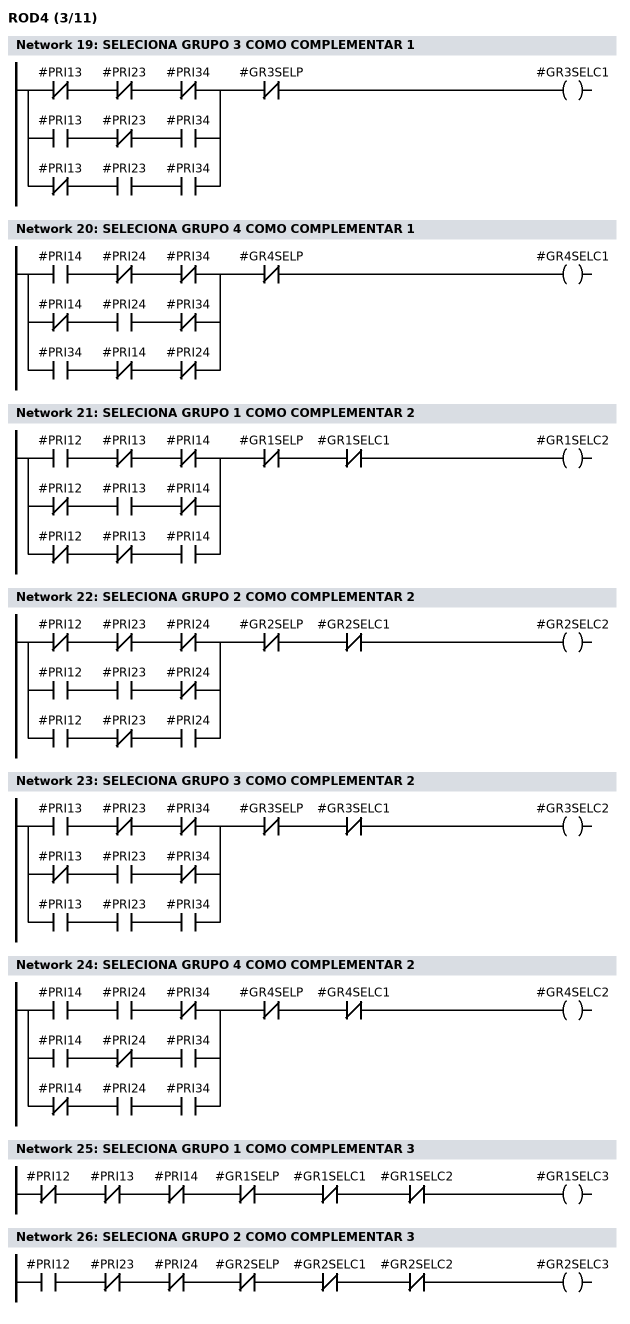
   RUNG wire#powerrail
      I_Contact( #PRI13 )
      I_Contact( #PRI23 )
      I_Contact( #PRI34 )
      wire#w1
      I_Contact( #GR3SELP )
      Coil( #GR3SELC1 )
   END_RUNG
   RUNG wire#powerrail
      Contact( #PRI13 )
      I_Contact( #PRI23 )
      Contact( #PRI34 )
   END_RUNG wire#w1
   RUNG wire#powerrail
      I_Contact( #PRI13 )
      Contact( #PRI23 )
      Contact( #PRI34 )
   END_RUNG wire#w1
   // the same network as SCL:
   #GR3SELC1 := ((NOT #PRI13 AND NOT #PRI23 AND NOT #PRI34) OR (#PRI13 AND NOT #PRI23 AND #PRI34) OR (NOT #PRI13 AND #PRI23 AND #PRI34)) AND NOT #GR3SELP;
END_REGION

REGION Network 20: SELECIONA GRUPO 4 COMO COMPLEMENTAR 1
   RUNG wire#powerrail
      Contact( #PRI14 )
      I_Contact( #PRI24 )
      I_Contact( #PRI34 )
      wire#w1
      I_Contact( #GR4SELP )
      Coil( #GR4SELC1 )
   END_RUNG
   RUNG wire#powerrail
      I_Contact( #PRI14 )
      Contact( #PRI24 )
      I_Contact( #PRI34 )
   END_RUNG wire#w1
   RUNG wire#powerrail
      Contact( #PRI34 )
      I_Contact( #PRI14 )
      I_Contact( #PRI24 )
   END_RUNG wire#w1
   // the same network as SCL:
   #GR4SELC1 := ((#PRI14 AND NOT #PRI24 AND NOT #PRI34) OR (NOT #PRI14 AND #PRI24 AND NOT #PRI34) OR (#PRI34 AND NOT #PRI14 AND NOT #PRI24)) AND NOT #GR4SELP;
END_REGION

REGION Network 21: SELECIONA GRUPO 1 COMO COMPLEMENTAR 2
   RUNG wire#powerrail
      Contact( #PRI12 )
      I_Contact( #PRI13 )
      I_Contact( #PRI14 )
      wire#w1
      I_Contact( #GR1SELP )
      I_Contact( #GR1SELC1 )
      Coil( #GR1SELC2 )
   END_RUNG
   RUNG wire#powerrail
      I_Contact( #PRI12 )
      Contact( #PRI13 )
      I_Contact( #PRI14 )
   END_RUNG wire#w1
   RUNG wire#powerrail
      I_Contact( #PRI12 )
      I_Contact( #PRI13 )
      Contact( #PRI14 )
   END_RUNG wire#w1
   // the same network as SCL:
   #GR1SELC2 := ((#PRI12 AND NOT #PRI13 AND NOT #PRI14) OR (NOT #PRI12 AND #PRI13 AND NOT #PRI14) OR (NOT #PRI12 AND NOT #PRI13 AND #PRI14)) AND NOT #GR1SELP AND NOT #GR1SELC1;
END_REGION

REGION Network 22: SELECIONA GRUPO 2 COMO COMPLEMENTAR 2
   RUNG wire#powerrail
      I_Contact( #PRI12 )
      I_Contact( #PRI23 )
      I_Contact( #PRI24 )
      wire#w1
      I_Contact( #GR2SELP )
      I_Contact( #GR2SELC1 )
      Coil( #GR2SELC2 )
   END_RUNG
   RUNG wire#powerrail
      Contact( #PRI12 )
      Contact( #PRI23 )
      I_Contact( #PRI24 )
   END_RUNG wire#w1
   RUNG wire#powerrail
      Contact( #PRI12 )
      I_Contact( #PRI23 )
      Contact( #PRI24 )
   END_RUNG wire#w1
   // the same network as SCL:
   #GR2SELC2 := ((NOT #PRI12 AND NOT #PRI23 AND NOT #PRI24) OR (#PRI12 AND #PRI23 AND NOT #PRI24) OR (#PRI12 AND NOT #PRI23 AND #PRI24)) AND NOT #GR2SELP AND NOT #GR2SELC1;
END_REGION

REGION Network 23: SELECIONA GRUPO 3 COMO COMPLEMENTAR 2
   RUNG wire#powerrail
      Contact( #PRI13 )
      I_Contact( #PRI23 )
      I_Contact( #PRI34 )
      wire#w1
      I_Contact( #GR3SELP )
      I_Contact( #GR3SELC1 )
      Coil( #GR3SELC2 )
   END_RUNG
   RUNG wire#powerrail
      I_Contact( #PRI13 )
      Contact( #PRI23 )
      I_Contact( #PRI34 )
   END_RUNG wire#w1
   RUNG wire#powerrail
      Contact( #PRI13 )
      Contact( #PRI23 )
      Contact( #PRI34 )
   END_RUNG wire#w1
   // the same network as SCL:
   #GR3SELC2 := ((#PRI13 AND NOT #PRI23 AND NOT #PRI34) OR (NOT #PRI13 AND #PRI23 AND NOT #PRI34) OR (#PRI13 AND #PRI23 AND #PRI34)) AND NOT #GR3SELP AND NOT #GR3SELC1;
END_REGION

REGION Network 24: SELECIONA GRUPO 4 COMO COMPLEMENTAR 2
   RUNG wire#powerrail
      Contact( #PRI14 )
      Contact( #PRI24 )
      I_Contact( #PRI34 )
      wire#w1
      I_Contact( #GR4SELP )
      I_Contact( #GR4SELC1 )
      Coil( #GR4SELC2 )
   END_RUNG
   RUNG wire#powerrail
      Contact( #PRI14 )
      I_Contact( #PRI24 )
      Contact( #PRI34 )
   END_RUNG wire#w1
   RUNG wire#powerrail
      I_Contact( #PRI14 )
      Contact( #PRI24 )
      Contact( #PRI34 )
   END_RUNG wire#w1
   // the same network as SCL:
   #GR4SELC2 := ((#PRI14 AND #PRI24 AND NOT #PRI34) OR (#PRI14 AND NOT #PRI24 AND #PRI34) OR (NOT #PRI14 AND #PRI24 AND #PRI34)) AND NOT #GR4SELP AND NOT #GR4SELC1;
END_REGION

REGION Network 25: SELECIONA GRUPO 1 COMO COMPLEMENTAR 3
   RUNG wire#powerrail
      I_Contact( #PRI12 )
      I_Contact( #PRI13 )
      I_Contact( #PRI14 )
      I_Contact( #GR1SELP )
      I_Contact( #GR1SELC1 )
      I_Contact( #GR1SELC2 )
      Coil( #GR1SELC3 )
   END_RUNG
   // the same network as SCL:
   #GR1SELC3 := NOT #PRI12 AND NOT #PRI13 AND NOT #PRI14 AND NOT #GR1SELP AND NOT #GR1SELC1 AND NOT #GR1SELC2;
END_REGION

REGION Network 26: SELECIONA GRUPO 2 COMO COMPLEMENTAR 3
   RUNG wire#powerrail
      Contact( #PRI12 )
      I_Contact( #PRI23 )
      I_Contact( #PRI24 )
      I_Contact( #GR2SELP )
      I_Contact( #GR2SELC1 )
      I_Contact( #GR2SELC2 )
      Coil( #GR2SELC3 )
   END_RUNG
   // the same network as SCL:
   #GR2SELC3 := #PRI12 AND NOT #PRI23 AND NOT #PRI24 AND NOT #GR2SELP AND NOT #GR2SELC1 AND NOT #GR2SELC2;
END_REGION

REGION Network 27: SELECIONA GRUPO 3 COMO COMPLEMENTAR 3
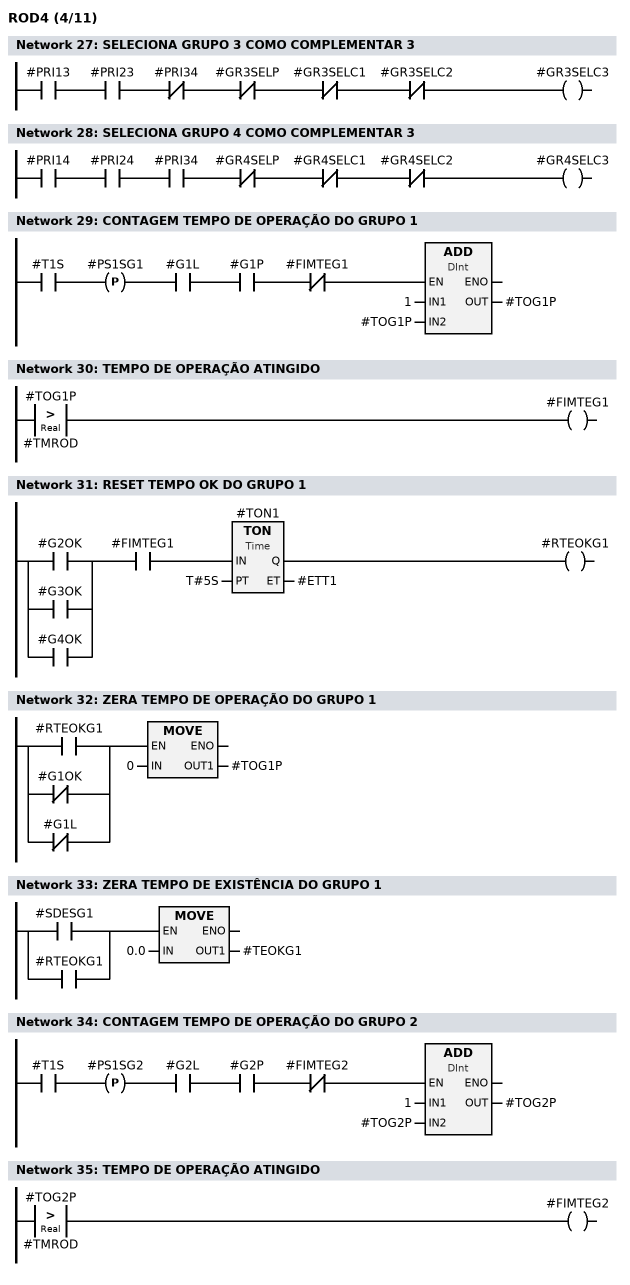
   RUNG wire#powerrail
      Contact( #PRI13 )
      Contact( #PRI23 )
      I_Contact( #PRI34 )
      I_Contact( #GR3SELP )
      I_Contact( #GR3SELC1 )
      I_Contact( #GR3SELC2 )
      Coil( #GR3SELC3 )
   END_RUNG
   // the same network as SCL:
   #GR3SELC3 := #PRI13 AND #PRI23 AND NOT #PRI34 AND NOT #GR3SELP AND NOT #GR3SELC1 AND NOT #GR3SELC2;
END_REGION

REGION Network 28: SELECIONA GRUPO 4 COMO COMPLEMENTAR 3
   RUNG wire#powerrail
      Contact( #PRI14 )
      Contact( #PRI24 )
      Contact( #PRI34 )
      I_Contact( #GR4SELP )
      I_Contact( #GR4SELC1 )
      I_Contact( #GR4SELC2 )
      Coil( #GR4SELC3 )
   END_RUNG
   // the same network as SCL:
   #GR4SELC3 := #PRI14 AND #PRI24 AND #PRI34 AND NOT #GR4SELP AND NOT #GR4SELC1 AND NOT #GR4SELC2;
END_REGION

REGION Network 29: CONTAGEM TEMPO DE OPERAÇÃO DO GRUPO 1
   RUNG wire#powerrail
      Contact( #T1S )
      P_Trig( #PS1SG1 )
      Contact( #G1L )
      Contact( #G1P )
      I_Contact( #FIMTEG1 )
      { S7_Templates := "SrcType := DInt"; S7_GenerateENO := "TRUE" } Add(in1 := 1, in2 := #TOG1P, out => #TOG1P)
   END_RUNG
   // the same network as SCL:
   #_w1 := #T1S AND NOT #PS1SG1;   // rising edge
   #PS1SG1 := #T1S;
   IF #_w1 AND #G1L AND #G1P AND NOT #FIMTEG1 THEN #TOG1P := 1 + #TOG1P; END_IF;
END_REGION

REGION Network 30: TEMPO DE OPERAÇÃO ATINGIDO
   RUNG wire#powerrail
      { S7_Templates := "SrcType := Real" } GT_Contact(in1 := #TOG1P, in2 := #TMROD)
      Coil( #FIMTEG1 )
   END_RUNG
   // the same network as SCL:
   #FIMTEG1 := #TOG1P > #TMROD;
END_REGION

REGION Network 31: RESET TEMPO OK DO GRUPO 1
   RUNG wire#powerrail
      Contact( #G2OK )
      wire#w1
      Contact( #FIMTEG1 )
      { S7_Templates := "time_type := Time" } #TON1.TON(pt := T#5S, et => #ETT1)
      Coil( #RTEOKG1 )
   END_RUNG
   RUNG wire#powerrail
      Contact( #G3OK )
   END_RUNG wire#w1
   RUNG wire#powerrail
      Contact( #G4OK )
   END_RUNG wire#w1
   // the same network as SCL:
   #TON1(IN := (#G2OK OR #G3OK OR #G4OK) AND #FIMTEG1, PT := T#5S, ET => #ETT1);   // TON
   #RTEOKG1 := #TON1.Q;
END_REGION

REGION Network 32: ZERA TEMPO DE OPERAÇÃO DO GRUPO 1
   RUNG wire#powerrail
      Contact( #RTEOKG1 )
      wire#w1
      { S7_GenerateENO := "TRUE" } Move(in := 0, out1 => #TOG1P)
   END_RUNG
   RUNG wire#powerrail
      I_Contact( #G1OK )
   END_RUNG wire#w1
   RUNG wire#powerrail
      I_Contact( #G1L )
   END_RUNG wire#w1
   // the same network as SCL:
   IF #RTEOKG1 OR NOT #G1OK OR NOT #G1L THEN #TOG1P := 0; END_IF;
END_REGION

REGION Network 33: ZERA TEMPO DE EXISTÊNCIA DO GRUPO 1
   RUNG wire#powerrail
      Contact( #SDESG1 )
      wire#w1
      { S7_GenerateENO := "TRUE" } Move(in := 0.0, out1 => #TEOKG1)
   END_RUNG
   RUNG wire#powerrail
      Contact( #RTEOKG1 )
   END_RUNG wire#w1
   // the same network as SCL:
   IF #SDESG1 OR #RTEOKG1 THEN #TEOKG1 := 0.0; END_IF;
END_REGION

REGION Network 34: CONTAGEM TEMPO DE OPERAÇÃO DO GRUPO 2
   RUNG wire#powerrail
      Contact( #T1S )
      P_Trig( #PS1SG2 )
      Contact( #G2L )
      Contact( #G2P )
      I_Contact( #FIMTEG2 )
      { S7_Templates := "SrcType := DInt"; S7_GenerateENO := "TRUE" } Add(in1 := 1, in2 := #TOG2P, out => #TOG2P)
   END_RUNG
   // the same network as SCL:
   #_w1 := #T1S AND NOT #PS1SG2;   // rising edge
   #PS1SG2 := #T1S;
   IF #_w1 AND #G2L AND #G2P AND NOT #FIMTEG2 THEN #TOG2P := 1 + #TOG2P; END_IF;
END_REGION

REGION Network 35: TEMPO DE OPERAÇÃO ATINGIDO
   RUNG wire#powerrail
      { S7_Templates := "SrcType := Real" } GT_Contact(in1 := #TOG2P, in2 := #TMROD)
      Coil( #FIMTEG2 )
   END_RUNG
   // the same network as SCL:
   #FIMTEG2 := #TOG2P > #TMROD;
END_REGION

REGION Network 36: RESET TEMPO OK DO GRUPO 2
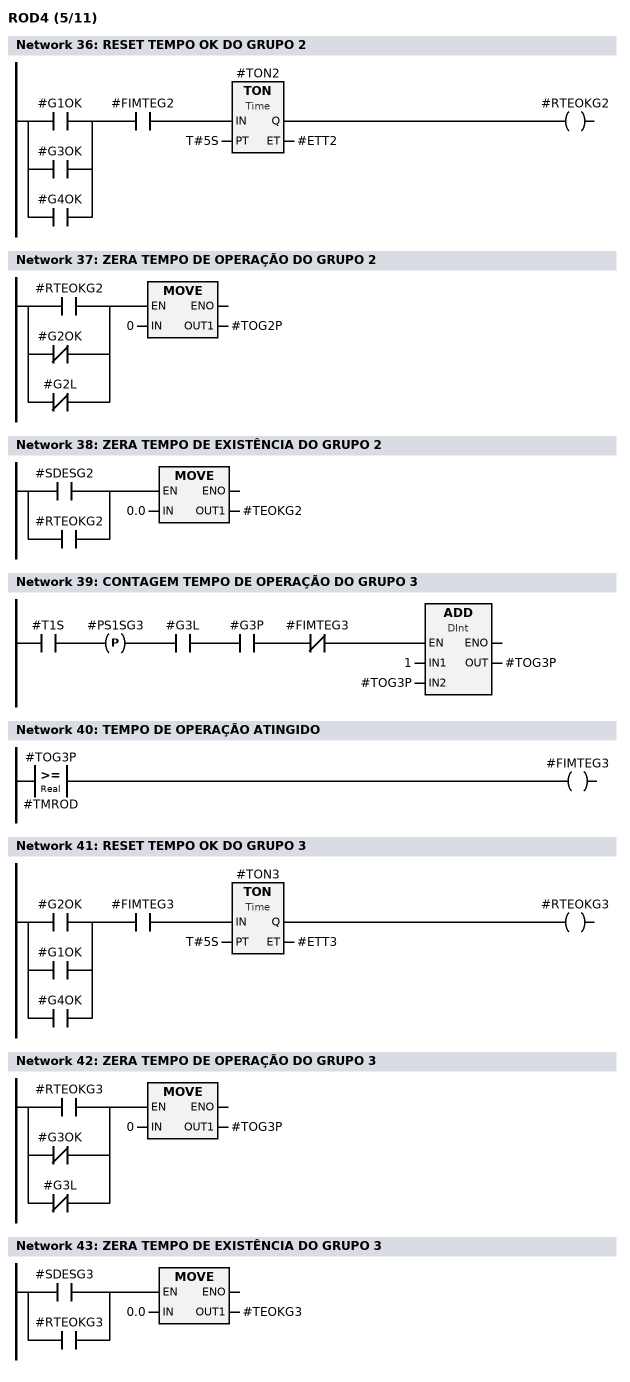
   RUNG wire#powerrail
      Contact( #G1OK )
      wire#w1
      Contact( #FIMTEG2 )
      { S7_Templates := "time_type := Time" } #TON2.TON(pt := T#5S, et => #ETT2)
      Coil( #RTEOKG2 )
   END_RUNG
   RUNG wire#powerrail
      Contact( #G3OK )
   END_RUNG wire#w1
   RUNG wire#powerrail
      Contact( #G4OK )
   END_RUNG wire#w1
   // the same network as SCL:
   #TON2(IN := (#G1OK OR #G3OK OR #G4OK) AND #FIMTEG2, PT := T#5S, ET => #ETT2);   // TON
   #RTEOKG2 := #TON2.Q;
END_REGION

REGION Network 37: ZERA TEMPO DE OPERAÇÃO DO GRUPO 2
   RUNG wire#powerrail
      Contact( #RTEOKG2 )
      wire#w1
      { S7_GenerateENO := "TRUE" } Move(in := 0, out1 => #TOG2P)
   END_RUNG
   RUNG wire#powerrail
      I_Contact( #G2OK )
   END_RUNG wire#w1
   RUNG wire#powerrail
      I_Contact( #G2L )
   END_RUNG wire#w1
   // the same network as SCL:
   IF #RTEOKG2 OR NOT #G2OK OR NOT #G2L THEN #TOG2P := 0; END_IF;
END_REGION

REGION Network 38: ZERA TEMPO DE EXISTÊNCIA DO GRUPO 2
   RUNG wire#powerrail
      Contact( #SDESG2 )
      wire#w1
      { S7_GenerateENO := "TRUE" } Move(in := 0.0, out1 => #TEOKG2)
   END_RUNG
   RUNG wire#powerrail
      Contact( #RTEOKG2 )
   END_RUNG wire#w1
   // the same network as SCL:
   IF #SDESG2 OR #RTEOKG2 THEN #TEOKG2 := 0.0; END_IF;
END_REGION

REGION Network 39: CONTAGEM TEMPO DE OPERAÇÃO DO GRUPO 3
   RUNG wire#powerrail
      Contact( #T1S )
      P_Trig( #PS1SG3 )
      Contact( #G3L )
      Contact( #G3P )
      I_Contact( #FIMTEG3 )
      { S7_Templates := "SrcType := DInt"; S7_GenerateENO := "TRUE" } Add(in1 := 1, in2 := #TOG3P, out => #TOG3P)
   END_RUNG
   // the same network as SCL:
   #_w1 := #T1S AND NOT #PS1SG3;   // rising edge
   #PS1SG3 := #T1S;
   IF #_w1 AND #G3L AND #G3P AND NOT #FIMTEG3 THEN #TOG3P := 1 + #TOG3P; END_IF;
END_REGION

REGION Network 40: TEMPO DE OPERAÇÃO ATINGIDO
   RUNG wire#powerrail
      { S7_Templates := "SrcType := Real" } GE_Contact(in1 := #TOG3P, in2 := #TMROD)
      Coil( #FIMTEG3 )
   END_RUNG
   // the same network as SCL:
   #FIMTEG3 := #TOG3P >= #TMROD;
END_REGION

REGION Network 41: RESET TEMPO OK DO GRUPO 3
   RUNG wire#powerrail
      Contact( #G2OK )
      wire#w1
      Contact( #FIMTEG3 )
      { S7_Templates := "time_type := Time" } #TON3.TON(pt := T#5S, et => #ETT3)
      Coil( #RTEOKG3 )
   END_RUNG
   RUNG wire#powerrail
      Contact( #G1OK )
   END_RUNG wire#w1
   RUNG wire#powerrail
      Contact( #G4OK )
   END_RUNG wire#w1
   // the same network as SCL:
   #TON3(IN := (#G2OK OR #G1OK OR #G4OK) AND #FIMTEG3, PT := T#5S, ET => #ETT3);   // TON
   #RTEOKG3 := #TON3.Q;
END_REGION

REGION Network 42: ZERA TEMPO DE OPERAÇÃO DO GRUPO 3
   RUNG wire#powerrail
      Contact( #RTEOKG3 )
      wire#w1
      { S7_GenerateENO := "TRUE" } Move(in := 0, out1 => #TOG3P)
   END_RUNG
   RUNG wire#powerrail
      I_Contact( #G3OK )
   END_RUNG wire#w1
   RUNG wire#powerrail
      I_Contact( #G3L )
   END_RUNG wire#w1
   // the same network as SCL:
   IF #RTEOKG3 OR NOT #G3OK OR NOT #G3L THEN #TOG3P := 0; END_IF;
END_REGION

REGION Network 43: ZERA TEMPO DE EXISTÊNCIA DO GRUPO 3
   RUNG wire#powerrail
      Contact( #SDESG3 )
      wire#w1
      { S7_GenerateENO := "TRUE" } Move(in := 0.0, out1 => #TEOKG3)
   END_RUNG
   RUNG wire#powerrail
      Contact( #RTEOKG3 )
   END_RUNG wire#w1
   // the same network as SCL:
   IF #SDESG3 OR #RTEOKG3 THEN #TEOKG3 := 0.0; END_IF;
END_REGION

REGION Network 44: CONTAGEM TEMPO DE OPERAÇÃO DO GRUPO 4
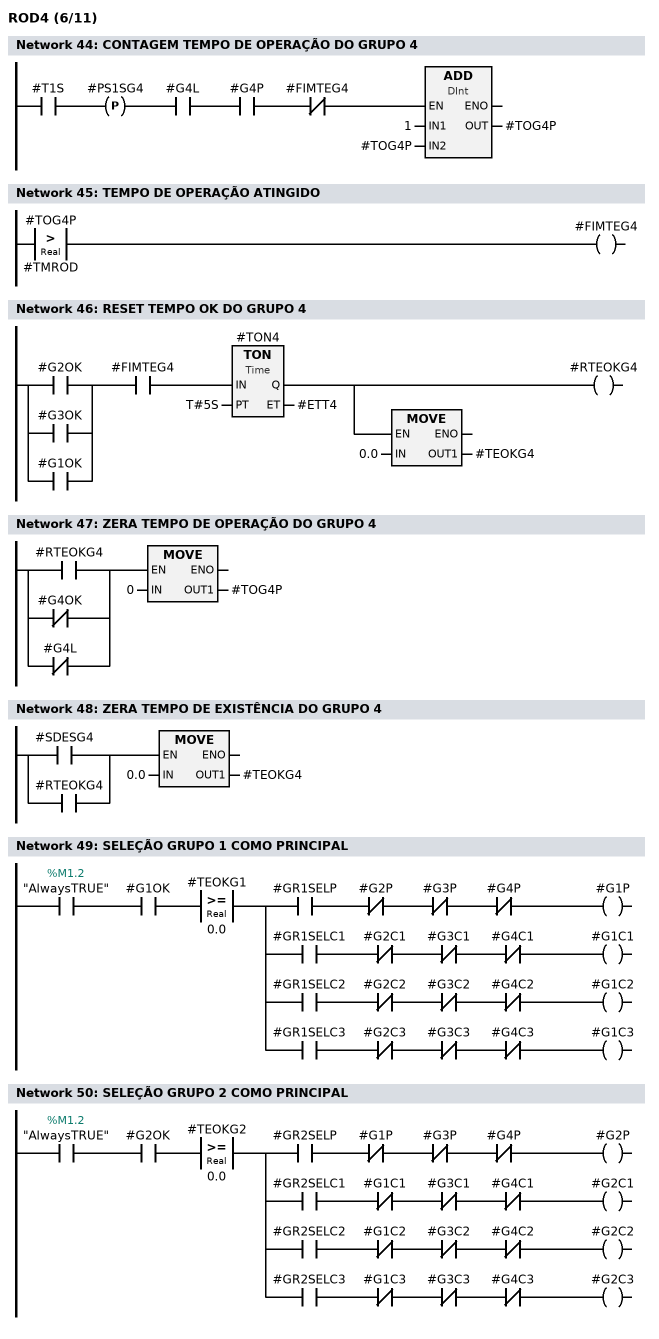
   RUNG wire#powerrail
      Contact( #T1S )
      P_Trig( #PS1SG4 )
      Contact( #G4L )
      Contact( #G4P )
      I_Contact( #FIMTEG4 )
      { S7_Templates := "SrcType := DInt"; S7_GenerateENO := "TRUE" } Add(in1 := 1, in2 := #TOG4P, out => #TOG4P)
   END_RUNG
   // the same network as SCL:
   #_w1 := #T1S AND NOT #PS1SG4;   // rising edge
   #PS1SG4 := #T1S;
   IF #_w1 AND #G4L AND #G4P AND NOT #FIMTEG4 THEN #TOG4P := 1 + #TOG4P; END_IF;
END_REGION

REGION Network 45: TEMPO DE OPERAÇÃO ATINGIDO
   RUNG wire#powerrail
      { S7_Templates := "SrcType := Real" } GT_Contact(in1 := #TOG4P, in2 := #TMROD)
      Coil( #FIMTEG4 )
   END_RUNG
   // the same network as SCL:
   #FIMTEG4 := #TOG4P > #TMROD;
END_REGION

REGION Network 46: RESET TEMPO OK DO GRUPO 4
   RUNG wire#powerrail
      Contact( #G2OK )
      wire#w1
      Contact( #FIMTEG4 )
      { S7_Templates := "time_type := Time" } #TON4.TON(pt := T#5S, et => #ETT4)
      wire#w2
      Coil( #RTEOKG4 )
   END_RUNG
   RUNG wire#powerrail
      Contact( #G3OK )
   END_RUNG wire#w1
   RUNG wire#powerrail
      Contact( #G1OK )
   END_RUNG wire#w1
   RUNG wire#w2
      { S7_GenerateENO := "TRUE" } Move(in := 0.0, out1 => #TEOKG4)
   END_RUNG
   // the same network as SCL:
   #TON4(IN := (#G2OK OR #G3OK OR #G1OK) AND #FIMTEG4, PT := T#5S, ET => #ETT4);   // TON
   #RTEOKG4 := #TON4.Q;
   IF #TON4.Q THEN #TEOKG4 := 0.0; END_IF;
END_REGION

REGION Network 47: ZERA TEMPO DE OPERAÇÃO DO GRUPO 4
   RUNG wire#powerrail
      Contact( #RTEOKG4 )
      wire#w1
      { S7_GenerateENO := "TRUE" } Move(in := 0, out1 => #TOG4P)
   END_RUNG
   RUNG wire#powerrail
      I_Contact( #G4OK )
   END_RUNG wire#w1
   RUNG wire#powerrail
      I_Contact( #G4L )
   END_RUNG wire#w1
   // the same network as SCL:
   IF #RTEOKG4 OR NOT #G4OK OR NOT #G4L THEN #TOG4P := 0; END_IF;
END_REGION

REGION Network 48: ZERA TEMPO DE EXISTÊNCIA DO GRUPO 4
   RUNG wire#powerrail
      Contact( #SDESG4 )
      wire#w1
      { S7_GenerateENO := "TRUE" } Move(in := 0.0, out1 => #TEOKG4)
   END_RUNG
   RUNG wire#powerrail
      Contact( #RTEOKG4 )
   END_RUNG wire#w1
   // the same network as SCL:
   IF #SDESG4 OR #RTEOKG4 THEN #TEOKG4 := 0.0; END_IF;
END_REGION

REGION Network 49: SELEÇÃO GRUPO 1 COMO PRINCIPAL
   RUNG wire#powerrail
      Contact( "AlwaysTRUE" )
      Contact( #G1OK )
      { S7_Templates := "SrcType := Real" } GE_Contact(in1 := #TEOKG1, in2 := 0.0)
      wire#w1
      Contact( #GR1SELP )
      I_Contact( #G2P )
      I_Contact( #G3P )
      I_Contact( #G4P )
      Coil( #G1P )
   END_RUNG
   RUNG wire#w1
      Contact( #GR1SELC1 )
      I_Contact( #G2C1 )
      I_Contact( #G3C1 )
      I_Contact( #G4C1 )
      Coil( #G1C1 )
   END_RUNG
   RUNG wire#w1
      Contact( #GR1SELC2 )
      I_Contact( #G2C2 )
      I_Contact( #G3C2 )
      I_Contact( #G4C2 )
      Coil( #G1C2 )
   END_RUNG
   RUNG wire#w1
      Contact( #GR1SELC3 )
      I_Contact( #G2C3 )
      I_Contact( #G3C3 )
      I_Contact( #G4C3 )
      Coil( #G1C3 )
   END_RUNG
   // the same network as SCL:
   #_w1 := "AlwaysTRUE" AND #G1OK AND (#TEOKG1 >= 0.0);
   #G1P := #_w1 AND #GR1SELP AND NOT #G2P AND NOT #G3P AND NOT #G4P;
   #G1C1 := #_w1 AND #GR1SELC1 AND NOT #G2C1 AND NOT #G3C1 AND NOT #G4C1;
   #G1C2 := #_w1 AND #GR1SELC2 AND NOT #G2C2 AND NOT #G3C2 AND NOT #G4C2;
   #G1C3 := #_w1 AND #GR1SELC3 AND NOT #G2C3 AND NOT #G3C3 AND NOT #G4C3;
END_REGION

REGION Network 50: SELEÇÃO GRUPO 2 COMO PRINCIPAL
   RUNG wire#powerrail
      Contact( "AlwaysTRUE" )
      Contact( #G2OK )
      { S7_Templates := "SrcType := Real" } GE_Contact(in1 := #TEOKG2, in2 := 0.0)
      wire#w1
      Contact( #GR2SELP )
      I_Contact( #G1P )
      I_Contact( #G3P )
      I_Contact( #G4P )
      Coil( #G2P )
   END_RUNG
   RUNG wire#w1
      Contact( #GR2SELC1 )
      I_Contact( #G1C1 )
      I_Contact( #G3C1 )
      I_Contact( #G4C1 )
      Coil( #G2C1 )
   END_RUNG
   RUNG wire#w1
      Contact( #GR2SELC2 )
      I_Contact( #G1C2 )
      I_Contact( #G3C2 )
      I_Contact( #G4C2 )
      Coil( #G2C2 )
   END_RUNG
   RUNG wire#w1
      Contact( #GR2SELC3 )
      I_Contact( #G1C3 )
      I_Contact( #G3C3 )
      I_Contact( #G4C3 )
      Coil( #G2C3 )
   END_RUNG
   // the same network as SCL:
   #_w1 := "AlwaysTRUE" AND #G2OK AND (#TEOKG2 >= 0.0);
   #G2P := #_w1 AND #GR2SELP AND NOT #G1P AND NOT #G3P AND NOT #G4P;
   #G2C1 := #_w1 AND #GR2SELC1 AND NOT #G1C1 AND NOT #G3C1 AND NOT #G4C1;
   #G2C2 := #_w1 AND #GR2SELC2 AND NOT #G1C2 AND NOT #G3C2 AND NOT #G4C2;
   #G2C3 := #_w1 AND #GR2SELC3 AND NOT #G1C3 AND NOT #G3C3 AND NOT #G4C3;
END_REGION

REGION Network 51: SELEÇÃO GRUPO 3 COMO PRINCIPAL
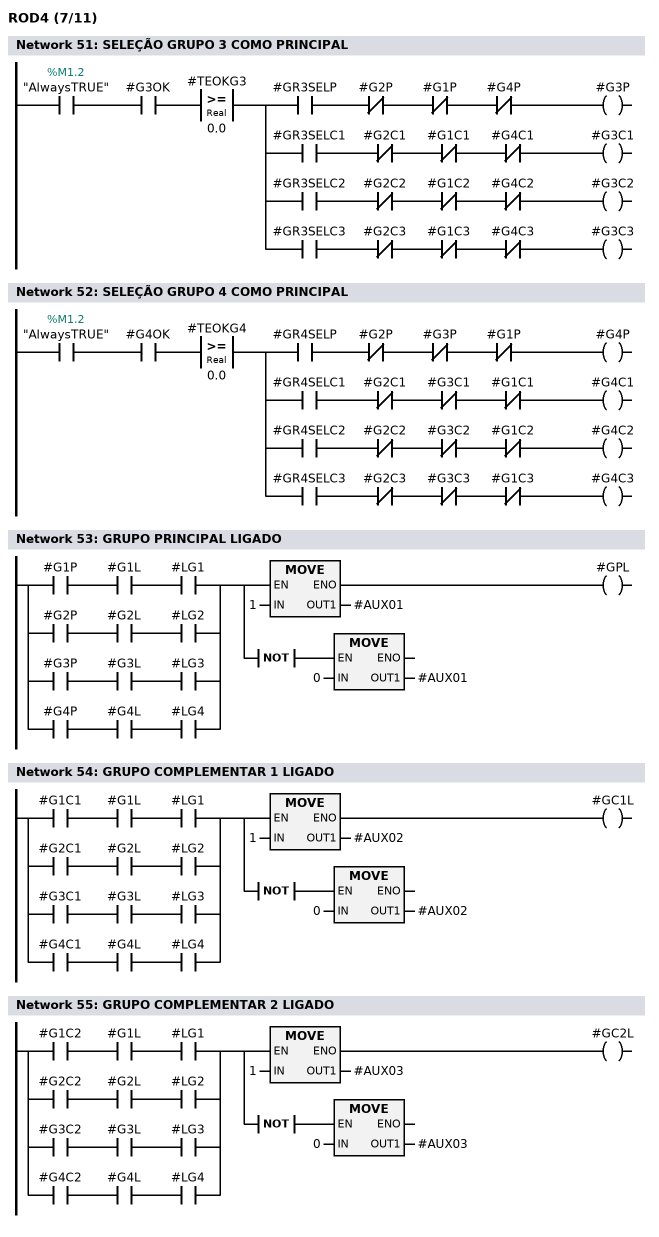
   RUNG wire#powerrail
      Contact( "AlwaysTRUE" )
      Contact( #G3OK )
      { S7_Templates := "SrcType := Real" } GE_Contact(in1 := #TEOKG3, in2 := 0.0)
      wire#w1
      Contact( #GR3SELP )
      I_Contact( #G2P )
      I_Contact( #G1P )
      I_Contact( #G4P )
      Coil( #G3P )
   END_RUNG
   RUNG wire#w1
      Contact( #GR3SELC1 )
      I_Contact( #G2C1 )
      I_Contact( #G1C1 )
      I_Contact( #G4C1 )
      Coil( #G3C1 )
   END_RUNG
   RUNG wire#w1
      Contact( #GR3SELC2 )
      I_Contact( #G2C2 )
      I_Contact( #G1C2 )
      I_Contact( #G4C2 )
      Coil( #G3C2 )
   END_RUNG
   RUNG wire#w1
      Contact( #GR3SELC3 )
      I_Contact( #G2C3 )
      I_Contact( #G1C3 )
      I_Contact( #G4C3 )
      Coil( #G3C3 )
   END_RUNG
   // the same network as SCL:
   #_w1 := "AlwaysTRUE" AND #G3OK AND (#TEOKG3 >= 0.0);
   #G3P := #_w1 AND #GR3SELP AND NOT #G2P AND NOT #G1P AND NOT #G4P;
   #G3C1 := #_w1 AND #GR3SELC1 AND NOT #G2C1 AND NOT #G1C1 AND NOT #G4C1;
   #G3C2 := #_w1 AND #GR3SELC2 AND NOT #G2C2 AND NOT #G1C2 AND NOT #G4C2;
   #G3C3 := #_w1 AND #GR3SELC3 AND NOT #G2C3 AND NOT #G1C3 AND NOT #G4C3;
END_REGION

REGION Network 52: SELEÇÃO GRUPO 4 COMO PRINCIPAL
   RUNG wire#powerrail
      Contact( "AlwaysTRUE" )
      Contact( #G4OK )
      { S7_Templates := "SrcType := Real" } GE_Contact(in1 := #TEOKG4, in2 := 0.0)
      wire#w1
      Contact( #GR4SELP )
      I_Contact( #G2P )
      I_Contact( #G3P )
      I_Contact( #G1P )
      Coil( #G4P )
   END_RUNG
   RUNG wire#w1
      Contact( #GR4SELC1 )
      I_Contact( #G2C1 )
      I_Contact( #G3C1 )
      I_Contact( #G1C1 )
      Coil( #G4C1 )
   END_RUNG
   RUNG wire#w1
      Contact( #GR4SELC2 )
      I_Contact( #G2C2 )
      I_Contact( #G3C2 )
      I_Contact( #G1C2 )
      Coil( #G4C2 )
   END_RUNG
   RUNG wire#w1
      Contact( #GR4SELC3 )
      I_Contact( #G2C3 )
      I_Contact( #G3C3 )
      I_Contact( #G1C3 )
      Coil( #G4C3 )
   END_RUNG
   // the same network as SCL:
   #_w1 := "AlwaysTRUE" AND #G4OK AND (#TEOKG4 >= 0.0);
   #G4P := #_w1 AND #GR4SELP AND NOT #G2P AND NOT #G3P AND NOT #G1P;
   #G4C1 := #_w1 AND #GR4SELC1 AND NOT #G2C1 AND NOT #G3C1 AND NOT #G1C1;
   #G4C2 := #_w1 AND #GR4SELC2 AND NOT #G2C2 AND NOT #G3C2 AND NOT #G1C2;
   #G4C3 := #_w1 AND #GR4SELC3 AND NOT #G2C3 AND NOT #G3C3 AND NOT #G1C3;
END_REGION

REGION Network 53: GRUPO PRINCIPAL LIGADO
   RUNG wire#powerrail
      Contact( #G1P )
      Contact( #G1L )
      Contact( #LG1 )
      wire#w1
      { S7_GenerateENO := "TRUE" } Move(in := 1, out1 => #AUX01)
      Coil( #GPL )
   END_RUNG
   RUNG wire#powerrail
      Contact( #G2P )
      Contact( #G2L )
      Contact( #LG2 )
   END_RUNG wire#w1
   RUNG wire#powerrail
      Contact( #G3P )
      Contact( #G3L )
      Contact( #LG3 )
   END_RUNG wire#w1
   RUNG wire#powerrail
      Contact( #G4P )
      Contact( #G4L )
      Contact( #LG4 )
   END_RUNG wire#w1
   RUNG wire#w1
      Not()
      { S7_GenerateENO := "TRUE" } Move(in := 0, out1 => #AUX01)
   END_RUNG
   // the same network as SCL:
   // ENO of a box is taken as its EN; it also drops when the box reports an error
   #_w1 := (#G1P AND #G1L AND #LG1) OR (#G2P AND #G2L AND #LG2) OR (#G3P AND #G3L AND #LG3) OR (#G4P AND #G4L AND #LG4);
   IF #_w1 THEN #AUX01 := 1; END_IF;
   #GPL := #_w1;
   IF NOT #_w1 THEN #AUX01 := 0; END_IF;
END_REGION

REGION Network 54: GRUPO COMPLEMENTAR 1 LIGADO
   RUNG wire#powerrail
      Contact( #G1C1 )
      Contact( #G1L )
      Contact( #LG1 )
      wire#w1
      { S7_GenerateENO := "TRUE" } Move(in := 1, out1 => #AUX02)
      Coil( #GC1L )
   END_RUNG
   RUNG wire#powerrail
      Contact( #G2C1 )
      Contact( #G2L )
      Contact( #LG2 )
   END_RUNG wire#w1
   RUNG wire#powerrail
      Contact( #G3C1 )
      Contact( #G3L )
      Contact( #LG3 )
   END_RUNG wire#w1
   RUNG wire#powerrail
      Contact( #G4C1 )
      Contact( #G4L )
      Contact( #LG4 )
   END_RUNG wire#w1
   RUNG wire#w1
      Not()
      { S7_GenerateENO := "TRUE" } Move(in := 0, out1 => #AUX02)
   END_RUNG
   // the same network as SCL:
   // ENO of a box is taken as its EN; it also drops when the box reports an error
   #_w1 := (#G1C1 AND #G1L AND #LG1) OR (#G2C1 AND #G2L AND #LG2) OR (#G3C1 AND #G3L AND #LG3) OR (#G4C1 AND #G4L AND #LG4);
   IF #_w1 THEN #AUX02 := 1; END_IF;
   #GC1L := #_w1;
   IF NOT #_w1 THEN #AUX02 := 0; END_IF;
END_REGION

REGION Network 55: GRUPO COMPLEMENTAR 2 LIGADO
   RUNG wire#powerrail
      Contact( #G1C2 )
      Contact( #G1L )
      Contact( #LG1 )
      wire#w1
      { S7_GenerateENO := "TRUE" } Move(in := 1, out1 => #AUX03)
      Coil( #GC2L )
   END_RUNG
   RUNG wire#powerrail
      Contact( #G2C2 )
      Contact( #G2L )
      Contact( #LG2 )
   END_RUNG wire#w1
   RUNG wire#powerrail
      Contact( #G3C2 )
      Contact( #G3L )
      Contact( #LG3 )
   END_RUNG wire#w1
   RUNG wire#powerrail
      Contact( #G4C2 )
      Contact( #G4L )
      Contact( #LG4 )
   END_RUNG wire#w1
   RUNG wire#w1
      Not()
      { S7_GenerateENO := "TRUE" } Move(in := 0, out1 => #AUX03)
   END_RUNG
   // the same network as SCL:
   // ENO of a box is taken as its EN; it also drops when the box reports an error
   #_w1 := (#G1C2 AND #G1L AND #LG1) OR (#G2C2 AND #G2L AND #LG2) OR (#G3C2 AND #G3L AND #LG3) OR (#G4C2 AND #G4L AND #LG4);
   IF #_w1 THEN #AUX03 := 1; END_IF;
   #GC2L := #_w1;
   IF NOT #_w1 THEN #AUX03 := 0; END_IF;
END_REGION

REGION Network 56: GRUPO COMPLEMENTAR 3 LIGADO
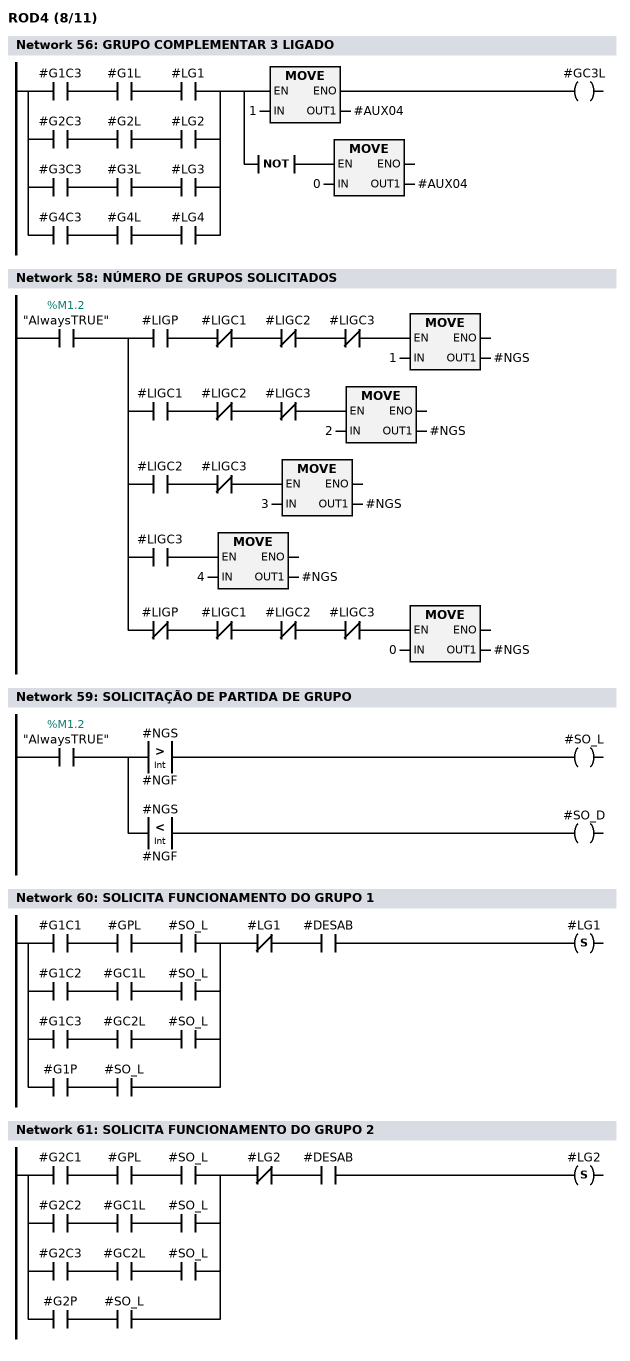
   RUNG wire#powerrail
      Contact( #G1C3 )
      Contact( #G1L )
      Contact( #LG1 )
      wire#w1
      { S7_GenerateENO := "TRUE" } Move(in := 1, out1 => #AUX04)
      Coil( #GC3L )
   END_RUNG
   RUNG wire#powerrail
      Contact( #G2C3 )
      Contact( #G2L )
      Contact( #LG2 )
   END_RUNG wire#w1
   RUNG wire#powerrail
      Contact( #G3C3 )
      Contact( #G3L )
      Contact( #LG3 )
   END_RUNG wire#w1
   RUNG wire#powerrail
      Contact( #G4C3 )
      Contact( #G4L )
      Contact( #LG4 )
   END_RUNG wire#w1
   RUNG wire#w1
      Not()
      { S7_GenerateENO := "TRUE" } Move(in := 0, out1 => #AUX04)
   END_RUNG
   // the same network as SCL:
   // ENO of a box is taken as its EN; it also drops when the box reports an error
   #_w1 := (#G1C3 AND #G1L AND #LG1) OR (#G2C3 AND #G2L AND #LG2) OR (#G3C3 AND #G3L AND #LG3) OR (#G4C3 AND #G4L AND #LG4);
   IF #_w1 THEN #AUX04 := 1; END_IF;
   #GC3L := #_w1;
   IF NOT #_w1 THEN #AUX04 := 0; END_IF;
END_REGION

NETWORK
TITLE = NÚMERO DE GRUPOS FUNCIONANDO

      L     #AUX01;
      L     #AUX02;
      +I;
      L     #AUX03;
      +I;
      L     #AUX04;
      +I;
      T     #NGF;

REGION Network 58: NÚMERO DE GRUPOS SOLICITADOS
   RUNG wire#powerrail
      Contact( "AlwaysTRUE" )
      wire#w1
      Contact( #LIGP )
      I_Contact( #LIGC1 )
      I_Contact( #LIGC2 )
      I_Contact( #LIGC3 )
      { S7_GenerateENO := "TRUE" } Move(in := 1, out1 => #NGS)
   END_RUNG
   RUNG wire#w1
      Contact( #LIGC1 )
      I_Contact( #LIGC2 )
      I_Contact( #LIGC3 )
      { S7_GenerateENO := "TRUE" } Move(in := 2, out1 => #NGS)
   END_RUNG
   RUNG wire#w1
      Contact( #LIGC2 )
      I_Contact( #LIGC3 )
      { S7_GenerateENO := "TRUE" } Move(in := 3, out1 => #NGS)
   END_RUNG
   RUNG wire#w1
      Contact( #LIGC3 )
      { S7_GenerateENO := "TRUE" } Move(in := 4, out1 => #NGS)
   END_RUNG
   RUNG wire#w1
      I_Contact( #LIGP )
      I_Contact( #LIGC1 )
      I_Contact( #LIGC2 )
      I_Contact( #LIGC3 )
      { S7_GenerateENO := "TRUE" } Move(in := 0, out1 => #NGS)
   END_RUNG
   // the same network as SCL:
   IF "AlwaysTRUE" AND #LIGP AND NOT #LIGC1 AND NOT #LIGC2 AND NOT #LIGC3 THEN #NGS := 1; END_IF;
   IF "AlwaysTRUE" AND #LIGC1 AND NOT #LIGC2 AND NOT #LIGC3 THEN #NGS := 2; END_IF;
   IF "AlwaysTRUE" AND #LIGC2 AND NOT #LIGC3 THEN #NGS := 3; END_IF;
   IF "AlwaysTRUE" AND #LIGC3 THEN #NGS := 4; END_IF;
   IF "AlwaysTRUE" AND NOT #LIGP AND NOT #LIGC1 AND NOT #LIGC2 AND NOT #LIGC3 THEN #NGS := 0; END_IF;
END_REGION

REGION Network 59: SOLICITAÇÃO DE PARTIDA DE GRUPO
   RUNG wire#powerrail
      Contact( "AlwaysTRUE" )
      wire#w1
      { S7_Templates := "SrcType := Int" } GT_Contact(in1 := #NGS, in2 := #NGF)
      Coil( #SO_L )
   END_RUNG
   RUNG wire#w1
      { S7_Templates := "SrcType := Int" } LT_Contact(in1 := #NGS, in2 := #NGF)
      Coil( #SO_D )
   END_RUNG
   // the same network as SCL:
   #SO_L := "AlwaysTRUE" AND (#NGS > #NGF);
   #SO_D := "AlwaysTRUE" AND (#NGS < #NGF);
END_REGION

REGION Network 60: SOLICITA FUNCIONAMENTO DO GRUPO 1
   RUNG wire#powerrail
      Contact( #G1C1 )
      Contact( #GPL )
      Contact( #SO_L )
      wire#w1
      I_Contact( #LG1 )
      Contact( #DESAB )
      S_Coil( #LG1 )
   END_RUNG
   RUNG wire#powerrail
      Contact( #G1C2 )
      Contact( #GC1L )
      Contact( #SO_L )
   END_RUNG wire#w1
   RUNG wire#powerrail
      Contact( #G1C3 )
      Contact( #GC2L )
      Contact( #SO_L )
   END_RUNG wire#w1
   RUNG wire#powerrail
      Contact( #G1P )
      Contact( #SO_L )
   END_RUNG wire#w1
   // the same network as SCL:
   IF ((#G1C1 AND #GPL AND #SO_L) OR (#G1C2 AND #GC1L AND #SO_L) OR (#G1C3 AND #GC2L AND #SO_L) OR (#G1P AND #SO_L)) AND NOT #LG1 AND #DESAB THEN
       #LG1 := TRUE;
   END_IF;
END_REGION

REGION Network 61: SOLICITA FUNCIONAMENTO DO GRUPO 2
   RUNG wire#powerrail
      Contact( #G2C1 )
      Contact( #GPL )
      Contact( #SO_L )
      wire#w1
      I_Contact( #LG2 )
      Contact( #DESAB )
      S_Coil( #LG2 )
   END_RUNG
   RUNG wire#powerrail
      Contact( #G2C2 )
      Contact( #GC1L )
      Contact( #SO_L )
   END_RUNG wire#w1
   RUNG wire#powerrail
      Contact( #G2C3 )
      Contact( #GC2L )
      Contact( #SO_L )
   END_RUNG wire#w1
   RUNG wire#powerrail
      Contact( #G2P )
      Contact( #SO_L )
   END_RUNG wire#w1
   // the same network as SCL:
   IF ((#G2C1 AND #GPL AND #SO_L) OR (#G2C2 AND #GC1L AND #SO_L) OR (#G2C3 AND #GC2L AND #SO_L) OR (#G2P AND #SO_L)) AND NOT #LG2 AND #DESAB THEN
       #LG2 := TRUE;
   END_IF;
END_REGION

REGION Network 62: SOLICITA FUNCIONAMENTO DO GRUPO 3
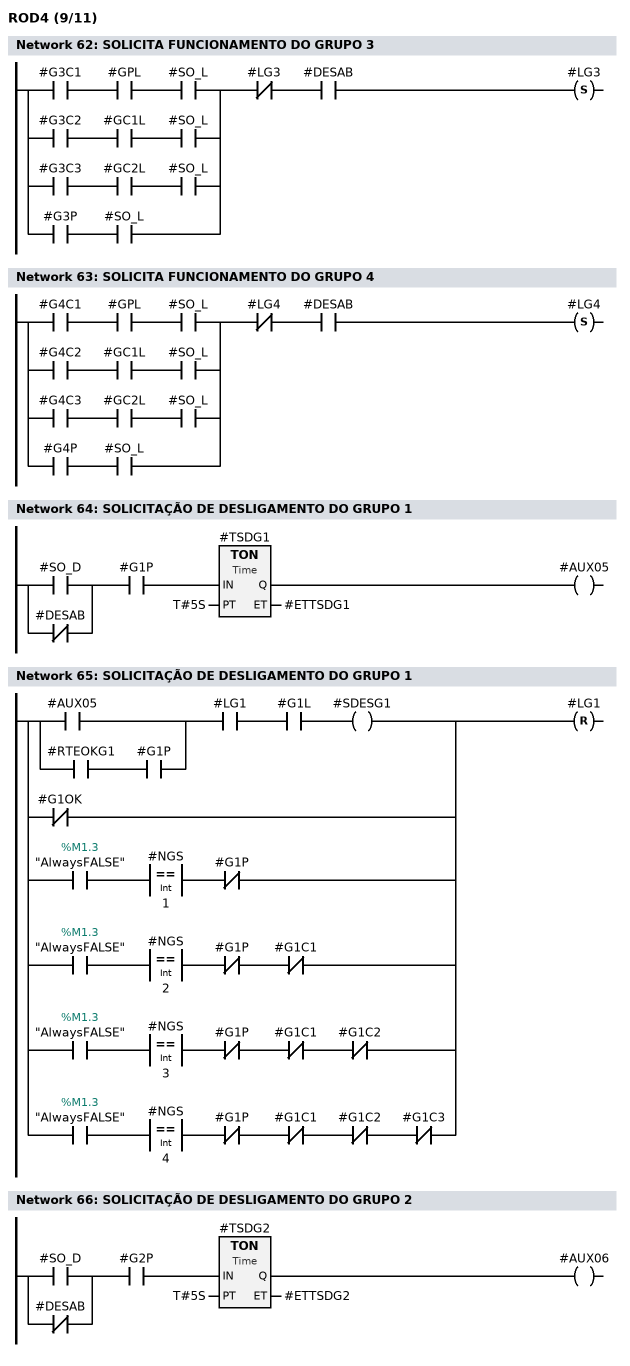
   RUNG wire#powerrail
      Contact( #G3C1 )
      Contact( #GPL )
      Contact( #SO_L )
      wire#w1
      I_Contact( #LG3 )
      Contact( #DESAB )
      S_Coil( #LG3 )
   END_RUNG
   RUNG wire#powerrail
      Contact( #G3C2 )
      Contact( #GC1L )
      Contact( #SO_L )
   END_RUNG wire#w1
   RUNG wire#powerrail
      Contact( #G3C3 )
      Contact( #GC2L )
      Contact( #SO_L )
   END_RUNG wire#w1
   RUNG wire#powerrail
      Contact( #G3P )
      Contact( #SO_L )
   END_RUNG wire#w1
   // the same network as SCL:
   IF ((#G3C1 AND #GPL AND #SO_L) OR (#G3C2 AND #GC1L AND #SO_L) OR (#G3C3 AND #GC2L AND #SO_L) OR (#G3P AND #SO_L)) AND NOT #LG3 AND #DESAB THEN
       #LG3 := TRUE;
   END_IF;
END_REGION

REGION Network 63: SOLICITA FUNCIONAMENTO DO GRUPO 4
   RUNG wire#powerrail
      Contact( #G4C1 )
      Contact( #GPL )
      Contact( #SO_L )
      wire#w1
      I_Contact( #LG4 )
      Contact( #DESAB )
      S_Coil( #LG4 )
   END_RUNG
   RUNG wire#powerrail
      Contact( #G4C2 )
      Contact( #GC1L )
      Contact( #SO_L )
   END_RUNG wire#w1
   RUNG wire#powerrail
      Contact( #G4C3 )
      Contact( #GC2L )
      Contact( #SO_L )
   END_RUNG wire#w1
   RUNG wire#powerrail
      Contact( #G4P )
      Contact( #SO_L )
   END_RUNG wire#w1
   // the same network as SCL:
   IF ((#G4C1 AND #GPL AND #SO_L) OR (#G4C2 AND #GC1L AND #SO_L) OR (#G4C3 AND #GC2L AND #SO_L) OR (#G4P AND #SO_L)) AND NOT #LG4 AND #DESAB THEN
       #LG4 := TRUE;
   END_IF;
END_REGION

REGION Network 64: SOLICITAÇÃO DE DESLIGAMENTO DO GRUPO 1
   RUNG wire#powerrail
      Contact( #SO_D )
      wire#w1
      Contact( #G1P )
      { S7_Templates := "time_type := Time" } #TSDG1.TON(pt := T#5S, et => #ETTSDG1)
      Coil( #AUX05 )
   END_RUNG
   RUNG wire#powerrail
      I_Contact( #DESAB )
   END_RUNG wire#w1
   // the same network as SCL:
   #TSDG1(IN := (#SO_D OR NOT #DESAB) AND #G1P, PT := T#5S, ET => #ETTSDG1);   // TON
   #AUX05 := #TSDG1.Q;
END_REGION

REGION Network 65: SOLICITAÇÃO DE DESLIGAMENTO DO GRUPO 1
   RUNG wire#powerrail
      Contact( #AUX05 )
      wire#w1
      Contact( #LG1 )
      Contact( #G1L )
      Coil( #SDESG1 )
      wire#w2
      R_Coil( #LG1 )
   END_RUNG
   RUNG wire#powerrail
      Contact( #RTEOKG1 )
      Contact( #G1P )
   END_RUNG wire#w1
   RUNG wire#powerrail
      I_Contact( #G1OK )
   END_RUNG wire#w2
   RUNG wire#powerrail
      Contact( "AlwaysFALSE" )
      { S7_Templates := "SrcType := Int" } EQ_Contact(in1 := #NGS, in2 := 1)
      I_Contact( #G1P )
   END_RUNG wire#w2
   RUNG wire#powerrail
      Contact( "AlwaysFALSE" )
      { S7_Templates := "SrcType := Int" } EQ_Contact(in1 := #NGS, in2 := 2)
      I_Contact( #G1P )
      I_Contact( #G1C1 )
   END_RUNG wire#w2
   RUNG wire#powerrail
      Contact( "AlwaysFALSE" )
      { S7_Templates := "SrcType := Int" } EQ_Contact(in1 := #NGS, in2 := 3)
      I_Contact( #G1P )
      I_Contact( #G1C1 )
      I_Contact( #G1C2 )
   END_RUNG wire#w2
   RUNG wire#powerrail
      Contact( "AlwaysFALSE" )
      { S7_Templates := "SrcType := Int" } EQ_Contact(in1 := #NGS, in2 := 4)
      I_Contact( #G1P )
      I_Contact( #G1C1 )
      I_Contact( #G1C2 )
      I_Contact( #G1C3 )
   END_RUNG wire#w2
   // the same network as SCL:
   #SDESG1 := (#AUX05 OR (#RTEOKG1 AND #G1P)) AND #LG1 AND #G1L;
   IF #SDESG1 OR NOT #G1OK OR ("AlwaysFALSE" AND (#NGS = 1) AND NOT #G1P) OR ("AlwaysFALSE" AND (#NGS = 2) AND NOT #G1P AND NOT #G1C1) OR ("AlwaysFALSE" AND (#NGS = 3) AND NOT #G1P AND NOT #G1C1 AND NOT #G1C2) OR ("AlwaysFALSE" AND (#NGS = 4) AND NOT #G1P AND NOT #G1C1 AND NOT #G1C2 AND NOT #G1C3) THEN
       #LG1 := FALSE;
   END_IF;
END_REGION

REGION Network 66: SOLICITAÇÃO DE DESLIGAMENTO DO GRUPO 2
   RUNG wire#powerrail
      Contact( #SO_D )
      wire#w1
      Contact( #G2P )
      { S7_Templates := "time_type := Time" } #TSDG2.TON(pt := T#5S, et => #ETTSDG2)
      Coil( #AUX06 )
   END_RUNG
   RUNG wire#powerrail
      I_Contact( #DESAB )
   END_RUNG wire#w1
   // the same network as SCL:
   #TSDG2(IN := (#SO_D OR NOT #DESAB) AND #G2P, PT := T#5S, ET => #ETTSDG2);   // TON
   #AUX06 := #TSDG2.Q;
END_REGION

REGION Network 67: SOLICITAÇÃO DE DESLIGAMENTO DO GRUPO 2
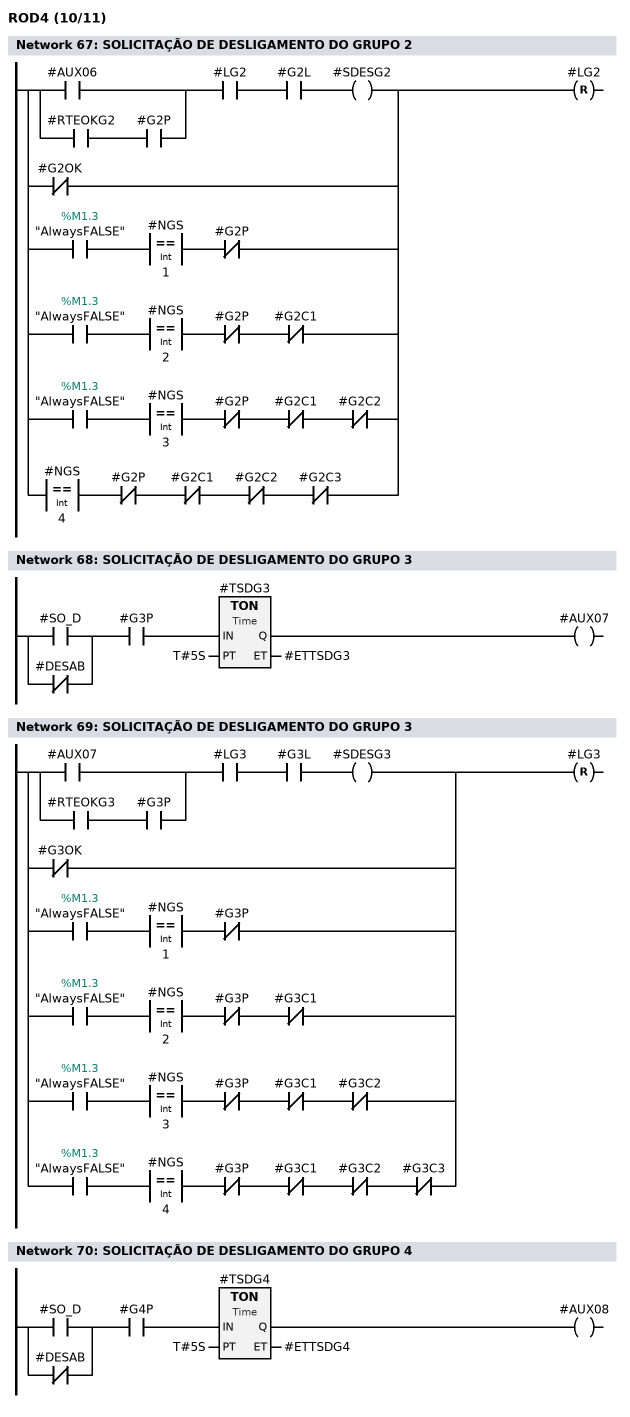
   RUNG wire#powerrail
      Contact( #AUX06 )
      wire#w1
      Contact( #LG2 )
      Contact( #G2L )
      Coil( #SDESG2 )
      wire#w2
      R_Coil( #LG2 )
   END_RUNG
   RUNG wire#powerrail
      Contact( #RTEOKG2 )
      Contact( #G2P )
   END_RUNG wire#w1
   RUNG wire#powerrail
      I_Contact( #G2OK )
   END_RUNG wire#w2
   RUNG wire#powerrail
      Contact( "AlwaysFALSE" )
      { S7_Templates := "SrcType := Int" } EQ_Contact(in1 := #NGS, in2 := 1)
      I_Contact( #G2P )
   END_RUNG wire#w2
   RUNG wire#powerrail
      Contact( "AlwaysFALSE" )
      { S7_Templates := "SrcType := Int" } EQ_Contact(in1 := #NGS, in2 := 2)
      I_Contact( #G2P )
      I_Contact( #G2C1 )
   END_RUNG wire#w2
   RUNG wire#powerrail
      Contact( "AlwaysFALSE" )
      { S7_Templates := "SrcType := Int" } EQ_Contact(in1 := #NGS, in2 := 3)
      I_Contact( #G2P )
      I_Contact( #G2C1 )
      I_Contact( #G2C2 )
   END_RUNG wire#w2
   RUNG wire#powerrail
      { S7_Templates := "SrcType := Int" } EQ_Contact(in1 := #NGS, in2 := 4)
      I_Contact( #G2P )
      I_Contact( #G2C1 )
      I_Contact( #G2C2 )
      I_Contact( #G2C3 )
   END_RUNG wire#w2
   // the same network as SCL:
   #SDESG2 := (#AUX06 OR (#RTEOKG2 AND #G2P)) AND #LG2 AND #G2L;
   IF #SDESG2 OR NOT #G2OK OR ("AlwaysFALSE" AND (#NGS = 1) AND NOT #G2P) OR ("AlwaysFALSE" AND (#NGS = 2) AND NOT #G2P AND NOT #G2C1) OR ("AlwaysFALSE" AND (#NGS = 3) AND NOT #G2P AND NOT #G2C1 AND NOT #G2C2) OR ((#NGS = 4) AND NOT #G2P AND NOT #G2C1 AND NOT #G2C2 AND NOT #G2C3) THEN
       #LG2 := FALSE;
   END_IF;
END_REGION

REGION Network 68: SOLICITAÇÃO DE DESLIGAMENTO DO GRUPO 3
   RUNG wire#powerrail
      Contact( #SO_D )
      wire#w1
      Contact( #G3P )
      { S7_Templates := "time_type := Time" } #TSDG3.TON(pt := T#5S, et => #ETTSDG3)
      Coil( #AUX07 )
   END_RUNG
   RUNG wire#powerrail
      I_Contact( #DESAB )
   END_RUNG wire#w1
   // the same network as SCL:
   #TSDG3(IN := (#SO_D OR NOT #DESAB) AND #G3P, PT := T#5S, ET => #ETTSDG3);   // TON
   #AUX07 := #TSDG3.Q;
END_REGION

REGION Network 69: SOLICITAÇÃO DE DESLIGAMENTO DO GRUPO 3
   RUNG wire#powerrail
      Contact( #AUX07 )
      wire#w1
      Contact( #LG3 )
      Contact( #G3L )
      Coil( #SDESG3 )
      wire#w2
      R_Coil( #LG3 )
   END_RUNG
   RUNG wire#powerrail
      Contact( #RTEOKG3 )
      Contact( #G3P )
   END_RUNG wire#w1
   RUNG wire#powerrail
      I_Contact( #G3OK )
   END_RUNG wire#w2
   RUNG wire#powerrail
      Contact( "AlwaysFALSE" )
      { S7_Templates := "SrcType := Int" } EQ_Contact(in1 := #NGS, in2 := 1)
      I_Contact( #G3P )
   END_RUNG wire#w2
   RUNG wire#powerrail
      Contact( "AlwaysFALSE" )
      { S7_Templates := "SrcType := Int" } EQ_Contact(in1 := #NGS, in2 := 2)
      I_Contact( #G3P )
      I_Contact( #G3C1 )
   END_RUNG wire#w2
   RUNG wire#powerrail
      Contact( "AlwaysFALSE" )
      { S7_Templates := "SrcType := Int" } EQ_Contact(in1 := #NGS, in2 := 3)
      I_Contact( #G3P )
      I_Contact( #G3C1 )
      I_Contact( #G3C2 )
   END_RUNG wire#w2
   RUNG wire#powerrail
      Contact( "AlwaysFALSE" )
      { S7_Templates := "SrcType := Int" } EQ_Contact(in1 := #NGS, in2 := 4)
      I_Contact( #G3P )
      I_Contact( #G3C1 )
      I_Contact( #G3C2 )
      I_Contact( #G3C3 )
   END_RUNG wire#w2
   // the same network as SCL:
   #SDESG3 := (#AUX07 OR (#RTEOKG3 AND #G3P)) AND #LG3 AND #G3L;
   IF #SDESG3 OR NOT #G3OK OR ("AlwaysFALSE" AND (#NGS = 1) AND NOT #G3P) OR ("AlwaysFALSE" AND (#NGS = 2) AND NOT #G3P AND NOT #G3C1) OR ("AlwaysFALSE" AND (#NGS = 3) AND NOT #G3P AND NOT #G3C1 AND NOT #G3C2) OR ("AlwaysFALSE" AND (#NGS = 4) AND NOT #G3P AND NOT #G3C1 AND NOT #G3C2 AND NOT #G3C3) THEN
       #LG3 := FALSE;
   END_IF;
END_REGION

REGION Network 70: SOLICITAÇÃO DE DESLIGAMENTO DO GRUPO 4
   RUNG wire#powerrail
      Contact( #SO_D )
      wire#w1
      Contact( #G4P )
      { S7_Templates := "time_type := Time" } #TSDG4.TON(pt := T#5S, et => #ETTSDG4)
      Coil( #AUX08 )
   END_RUNG
   RUNG wire#powerrail
      I_Contact( #DESAB )
   END_RUNG wire#w1
   // the same network as SCL:
   #TSDG4(IN := (#SO_D OR NOT #DESAB) AND #G4P, PT := T#5S, ET => #ETTSDG4);   // TON
   #AUX08 := #TSDG4.Q;
END_REGION

REGION Network 71: SOLICITAÇÃO DE DESLIGAMENTO DO GRUPO 4
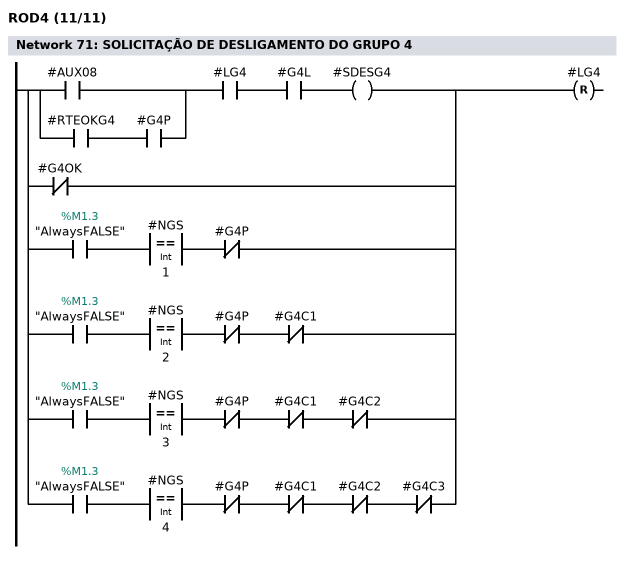
   RUNG wire#powerrail
      Contact( #AUX08 )
      wire#w1
      Contact( #LG4 )
      Contact( #G4L )
      Coil( #SDESG4 )
      wire#w2
      R_Coil( #LG4 )
   END_RUNG
   RUNG wire#powerrail
      Contact( #RTEOKG4 )
      Contact( #G4P )
   END_RUNG wire#w1
   RUNG wire#powerrail
      I_Contact( #G4OK )
   END_RUNG wire#w2
   RUNG wire#powerrail
      Contact( "AlwaysFALSE" )
      { S7_Templates := "SrcType := Int" } EQ_Contact(in1 := #NGS, in2 := 1)
      I_Contact( #G4P )
   END_RUNG wire#w2
   RUNG wire#powerrail
      Contact( "AlwaysFALSE" )
      { S7_Templates := "SrcType := Int" } EQ_Contact(in1 := #NGS, in2 := 2)
      I_Contact( #G4P )
      I_Contact( #G4C1 )
   END_RUNG wire#w2
   RUNG wire#powerrail
      Contact( "AlwaysFALSE" )
      { S7_Templates := "SrcType := Int" } EQ_Contact(in1 := #NGS, in2 := 3)
      I_Contact( #G4P )
      I_Contact( #G4C1 )
      I_Contact( #G4C2 )
   END_RUNG wire#w2
   RUNG wire#powerrail
      Contact( "AlwaysFALSE" )
      { S7_Templates := "SrcType := Int" } EQ_Contact(in1 := #NGS, in2 := 4)
      I_Contact( #G4P )
      I_Contact( #G4C1 )
      I_Contact( #G4C2 )
      I_Contact( #G4C3 )
   END_RUNG wire#w2
   // the same network as SCL:
   #SDESG4 := (#AUX08 OR (#RTEOKG4 AND #G4P)) AND #LG4 AND #G4L;
   IF #SDESG4 OR NOT #G4OK OR ("AlwaysFALSE" AND (#NGS = 1) AND NOT #G4P) OR ("AlwaysFALSE" AND (#NGS = 2) AND NOT #G4P AND NOT #G4C1) OR ("AlwaysFALSE" AND (#NGS = 3) AND NOT #G4P AND NOT #G4C1 AND NOT #G4C2) OR ("AlwaysFALSE" AND (#NGS = 4) AND NOT #G4P AND NOT #G4C1 AND NOT #G4C2 AND NOT #G4C3) THEN
       #LG4 := FALSE;
   END_IF;
END_REGION
END_FUNCTION_BLOCK

FUNCTION "AlARME" : Void   // FC3, LAD
{ S7_Optimized_Access := 'TRUE' }
VERSION : 0.1
// stored: AutoNumber true, IsIECCheckEnabled false, SetENOAutomatically false, UDAEnableTagReadback false
BEGIN

REGION Network 1: ALARMES IHM
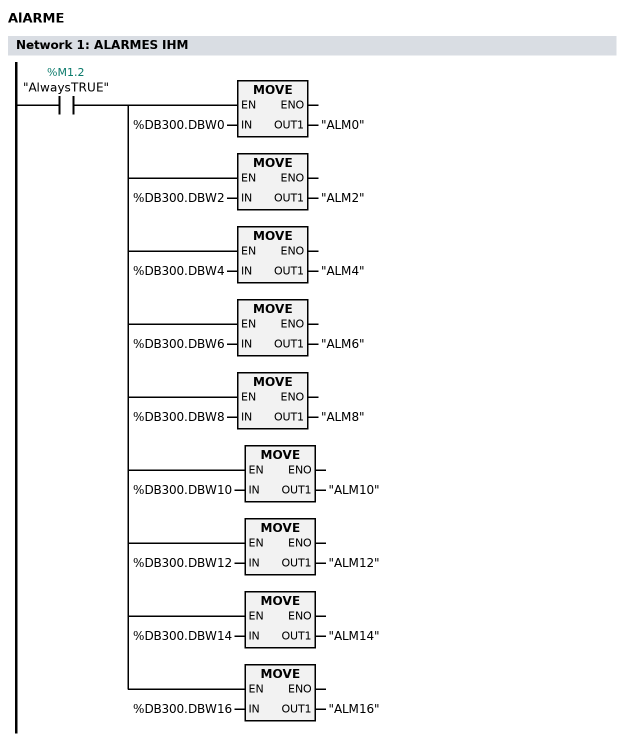
   RUNG wire#powerrail
      Contact( "AlwaysTRUE" )
      wire#w1
      Move(in := %DB300.DBW0, out1 => "ALM0")
   END_RUNG
   RUNG wire#w1
      Move(in := %DB300.DBW2, out1 => "ALM2")
   END_RUNG
   RUNG wire#w1
      Move(in := %DB300.DBW4, out1 => "ALM4")
   END_RUNG
   RUNG wire#w1
      Move(in := %DB300.DBW6, out1 => "ALM6")
   END_RUNG
   RUNG wire#w1
      Move(in := %DB300.DBW8, out1 => "ALM8")
   END_RUNG
   RUNG wire#w1
      Move(in := %DB300.DBW10, out1 => "ALM10")
   END_RUNG
   RUNG wire#w1
      Move(in := %DB300.DBW12, out1 => "ALM12")
   END_RUNG
   RUNG wire#w1
      Move(in := %DB300.DBW14, out1 => "ALM14")
   END_RUNG
   RUNG wire#w1
      Move(in := %DB300.DBW16, out1 => "ALM16")
   END_RUNG
   // the same network as SCL:
   IF "AlwaysTRUE" THEN
       "ALM0" := %DB300.DBW0;
       "ALM2" := %DB300.DBW2;
       "ALM4" := %DB300.DBW4;
       "ALM6" := %DB300.DBW6;
       "ALM8" := %DB300.DBW8;
       "ALM10" := %DB300.DBW10;
       "ALM12" := %DB300.DBW12;
       "ALM14" := %DB300.DBW14;
       "ALM16" := %DB300.DBW16;
   END_IF;
END_REGION
END_FUNCTION

FUNCTION_BLOCK "teste"   // FB1, SCL
{ S7_Optimized_Access := 'TRUE' }
VERSION : 0.1
// stored: AutoNumber true, IsIECCheckEnabled false, IsRetainMemResEnabled false, MemoryReserve 100, SetENOAutomatically false, UDAEnableTagReadback false
   VAR
      tag1 : Int;
      tag2 : Int;
      tag3 : Int;
   END_VAR
BEGIN

   #tag1 := 0;


   WHILE #tag1 < 100 DO
       #tag1 := #tag1 + 1;
           IF #tag1 >= 99 THEN
               #tag1 := 0;
           END_IF;// Statement section WHILE
   END_WHILE;
END_FUNCTION_BLOCK

ORGANIZATION_BLOCK "CYC_INT5"   // OB35, LAD, CyclicInterrupt
TITLE = CONTROLE DE PID
{ S7_Optimized_Access := 'FALSE' }
VERSION : 0.1
// stored: AutoNumber false, IsIECCheckEnabled false, SetENOAutomatically false
   VAR_TEMP
      OB35_EV_CLASS : Byte;
      OB35_STRT_INF : Byte;
      OB35_PRIORITY : Byte;
      OB35_OB_NUMBR : Byte;
      OB35_RESERVED_1 : Byte;
      OB35_RESERVED_2 : Byte;
      OB35_PHASE_OFFSET : Word;
      OB35_RESERVED_3 : Int;
      OB35_EXC_FREQ : Int;
      OB35_DATE_TIME : Date_And_Time;
      "SPM-EEEB" : Real;   // Setpoint manual PID tanque de aeração 1
      EEEB_IT : Time;   // Ajuste integral do PID
      EEEB_DT : Time;   // Ajuste derivativo do PID
      EEEB_AUX : Real;   // Setpoint manual PID - auxiliar
      EEEB_P : Real;   // Setpoint manual PID - auxiliar
   END_VAR
   VAR_TEMP   // added for the SCL form of the ladder/FBD networks
      _w1 : Bool;
      _w2 : Bool;
      _w3 : Bool;
      _w4 : Bool;
   END_VAR
BEGIN

NETWORK
TITLE = CONVERSÃO DOS SETPOINTS PARA TEMPO PID EEEB


//CONVERSÃO DOS SETPOINTS DE TEMPO PID EEEB
      L     "PID"."PID-EEEB-I";
      L     1000.0;
      *R;
      RND;
      T     #EEEB_IT;

      L     "PID"."PID-EEEB-D";
      L     1000.0;
      *R;
      RND;
      T     #EEEB_DT;

      L     "PID"."PID-EEEB-P";
      L     -1.0;
      *R;
      T     #EEEB_P;


REGION Network 2: PID TANQUE DE AERAÇÃO 1
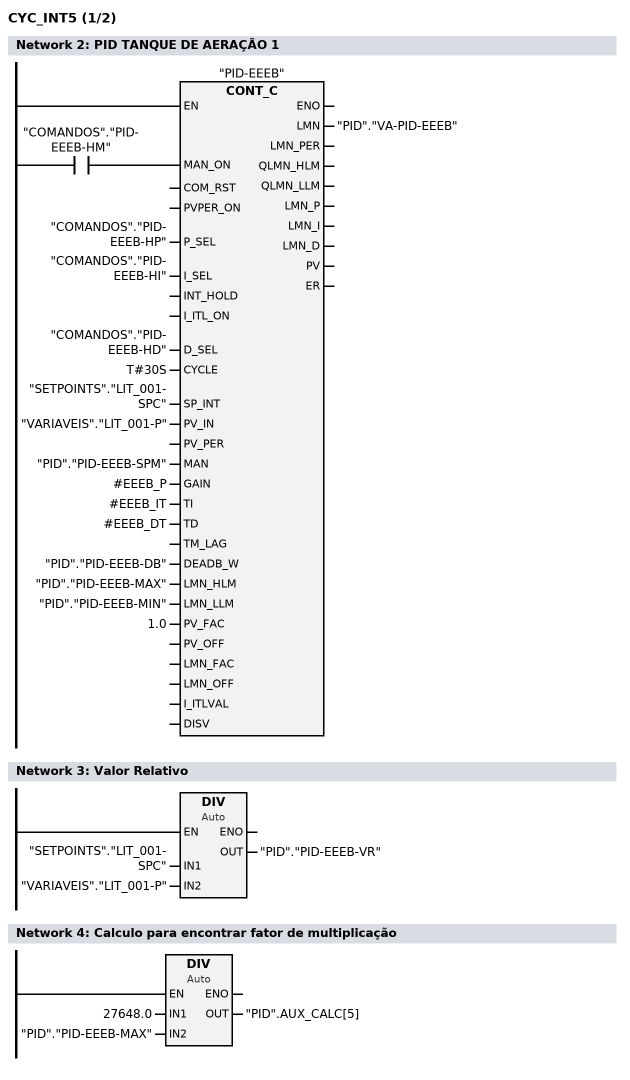
   RUNG wire#powerrail
      "PID-EEEB".CONT_C(MAN_ON := wire#w1, COM_RST :=, PVPER_ON :=, P_SEL := "COMANDOS"."PID-EEEB-HP", I_SEL := "COMANDOS"."PID-EEEB-HI", INT_HOLD :=, I_ITL_ON :=, D_SEL := "COMANDOS"."PID-EEEB-HD", CYCLE := T#30S, SP_INT := "SETPOINTS"."LIT_001-SPC", PV_IN := "VARIAVEIS"."LIT_001-P", PV_PER :=, MAN := "PID"."PID-EEEB-SPM", GAIN := #EEEB_P, TI := #EEEB_IT, TD := #EEEB_DT, TM_LAG :=, DEADB_W := "PID"."PID-EEEB-DB", LMN_HLM := "PID"."PID-EEEB-MAX", LMN_LLM := "PID"."PID-EEEB-MIN", PV_FAC := 1.0, PV_OFF :=, LMN_FAC :=, LMN_OFF :=, I_ITLVAL :=, DISV :=, LMN => "PID"."VA-PID-EEEB", LMN_PER =>, QLMN_HLM =>, QLMN_LLM =>, LMN_P =>, LMN_I =>, LMN_D =>, PV =>, ER =>)
   END_RUNG
   RUNG wire#powerrail
      Contact( "COMANDOS"."PID-EEEB-HM" )
   END_RUNG wire#w1
   // the same network as SCL:
   "PID-EEEB"(MAN_ON := "COMANDOS"."PID-EEEB-HM",   // CONT_C
              P_SEL := "COMANDOS"."PID-EEEB-HP",
              I_SEL := "COMANDOS"."PID-EEEB-HI",
              D_SEL := "COMANDOS"."PID-EEEB-HD",
              CYCLE := T#30S,
              SP_INT := "SETPOINTS"."LIT_001-SPC",
              PV_IN := "VARIAVEIS"."LIT_001-P",
              MAN := "PID"."PID-EEEB-SPM",
              GAIN := #EEEB_P,
              TI := #EEEB_IT,
              TD := #EEEB_DT,
              DEADB_W := "PID"."PID-EEEB-DB",
              LMN_HLM := "PID"."PID-EEEB-MAX",
              LMN_LLM := "PID"."PID-EEEB-MIN",
              PV_FAC := 1.0,
              LMN => "PID"."VA-PID-EEEB");
END_REGION

REGION Network 3: Valor Relativo
   RUNG wire#powerrail
      Div(in1 := "SETPOINTS"."LIT_001-SPC", in2 := "VARIAVEIS"."LIT_001-P", out => "PID"."PID-EEEB-VR")
   END_RUNG
   // the same network as SCL:
   "PID"."PID-EEEB-VR" := "SETPOINTS"."LIT_001-SPC" / "VARIAVEIS"."LIT_001-P";
END_REGION

REGION Network 4: Calculo para encontrar fator de multiplicação
   RUNG wire#powerrail
      Div(in1 := 27648.0, in2 := "PID"."PID-EEEB-MAX", out => "PID".AUX_CALC[5])
   END_RUNG
   // the same network as SCL:
   "PID".AUX_CALC[5] := 27648.0 / "PID"."PID-EEEB-MAX";
END_REGION

REGION Network 5: Movimenta saida PID para entrada analógica inversor
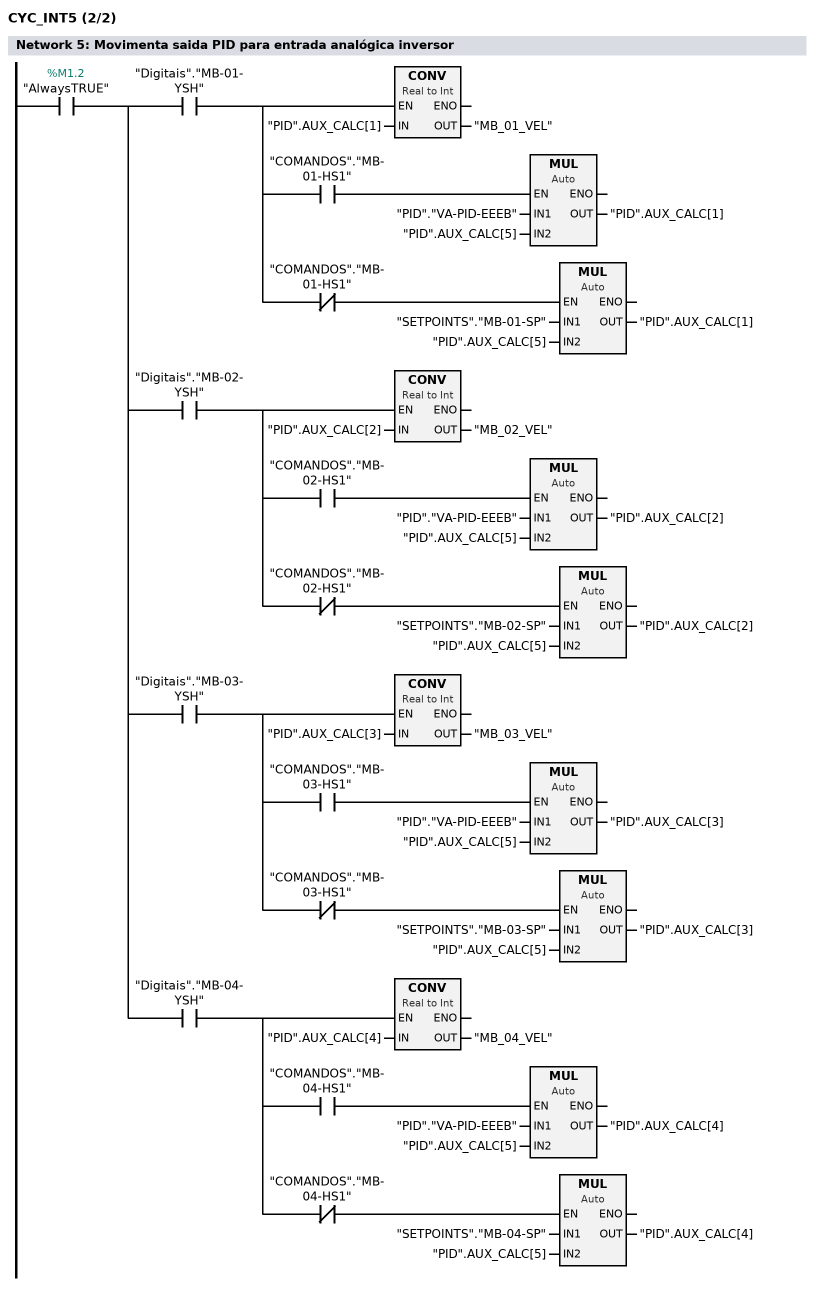
   RUNG wire#powerrail
      Contact( "AlwaysTRUE" )
      wire#w1
      Contact( "Digitais"."MB-01-YSH" )
      wire#w2
      { S7_Templates := "[SrcType := Real, DestType := Int]" } Convert(in := "PID".AUX_CALC[1], out => "MB_01_VEL")
   END_RUNG
   RUNG wire#w2
      Contact( "COMANDOS"."MB-01-HS1" )
      Mul(in1 := "PID"."VA-PID-EEEB", in2 := "PID".AUX_CALC[5], out => "PID".AUX_CALC[1])
   END_RUNG
   RUNG wire#w2
      I_Contact( "COMANDOS"."MB-01-HS1" )
      Mul(in1 := "SETPOINTS"."MB-01-SP", in2 := "PID".AUX_CALC[5], out => "PID".AUX_CALC[1])
   END_RUNG
   RUNG wire#w1
      Contact( "Digitais"."MB-02-YSH" )
      wire#w3
      { S7_Templates := "[SrcType := Real, DestType := Int]" } Convert(in := "PID".AUX_CALC[2], out => "MB_02_VEL")
   END_RUNG
   RUNG wire#w3
      Contact( "COMANDOS"."MB-02-HS1" )
      Mul(in1 := "PID"."VA-PID-EEEB", in2 := "PID".AUX_CALC[5], out => "PID".AUX_CALC[2])
   END_RUNG
   RUNG wire#w3
      I_Contact( "COMANDOS"."MB-02-HS1" )
      Mul(in1 := "SETPOINTS"."MB-02-SP", in2 := "PID".AUX_CALC[5], out => "PID".AUX_CALC[2])
   END_RUNG
   RUNG wire#w1
      Contact( "Digitais"."MB-03-YSH" )
      wire#w4
      { S7_Templates := "[SrcType := Real, DestType := Int]" } Convert(in := "PID".AUX_CALC[3], out => "MB_03_VEL")
   END_RUNG
   RUNG wire#w4
      Contact( "COMANDOS"."MB-03-HS1" )
      Mul(in1 := "PID"."VA-PID-EEEB", in2 := "PID".AUX_CALC[5], out => "PID".AUX_CALC[3])
   END_RUNG
   RUNG wire#w4
      I_Contact( "COMANDOS"."MB-03-HS1" )
      Mul(in1 := "SETPOINTS"."MB-03-SP", in2 := "PID".AUX_CALC[5], out => "PID".AUX_CALC[3])
   END_RUNG
   RUNG wire#w1
      Contact( "Digitais"."MB-04-YSH" )
      wire#w5
      { S7_Templates := "[SrcType := Real, DestType := Int]" } Convert(in := "PID".AUX_CALC[4], out => "MB_04_VEL")
   END_RUNG
   RUNG wire#w5
      Contact( "COMANDOS"."MB-04-HS1" )
      Mul(in1 := "PID"."VA-PID-EEEB", in2 := "PID".AUX_CALC[5], out => "PID".AUX_CALC[4])
   END_RUNG
   RUNG wire#w5
      I_Contact( "COMANDOS"."MB-04-HS1" )
      Mul(in1 := "SETPOINTS"."MB-04-SP", in2 := "PID".AUX_CALC[5], out => "PID".AUX_CALC[4])
   END_RUNG
   // the same network as SCL:
   #_w1 := "AlwaysTRUE" AND "Digitais"."MB-01-YSH";
   IF #_w1 THEN "MB_01_VEL" := REAL_TO_INT("PID".AUX_CALC[1]); END_IF;
   IF #_w1 AND "COMANDOS"."MB-01-HS1" THEN
       "PID".AUX_CALC[1] := "PID"."VA-PID-EEEB" * "PID".AUX_CALC[5];
   END_IF;
   IF #_w1 AND NOT "COMANDOS"."MB-01-HS1" THEN
       "PID".AUX_CALC[1] := "SETPOINTS"."MB-01-SP" * "PID".AUX_CALC[5];
   END_IF;
   #_w2 := "AlwaysTRUE" AND "Digitais"."MB-02-YSH";
   IF #_w2 THEN "MB_02_VEL" := REAL_TO_INT("PID".AUX_CALC[2]); END_IF;
   IF #_w2 AND "COMANDOS"."MB-02-HS1" THEN
       "PID".AUX_CALC[2] := "PID"."VA-PID-EEEB" * "PID".AUX_CALC[5];
   END_IF;
   IF #_w2 AND NOT "COMANDOS"."MB-02-HS1" THEN
       "PID".AUX_CALC[2] := "SETPOINTS"."MB-02-SP" * "PID".AUX_CALC[5];
   END_IF;
   #_w3 := "AlwaysTRUE" AND "Digitais"."MB-03-YSH";
   IF #_w3 THEN "MB_03_VEL" := REAL_TO_INT("PID".AUX_CALC[3]); END_IF;
   IF #_w3 AND "COMANDOS"."MB-03-HS1" THEN
       "PID".AUX_CALC[3] := "PID"."VA-PID-EEEB" * "PID".AUX_CALC[5];
   END_IF;
   IF #_w3 AND NOT "COMANDOS"."MB-03-HS1" THEN
       "PID".AUX_CALC[3] := "SETPOINTS"."MB-03-SP" * "PID".AUX_CALC[5];
   END_IF;
   #_w4 := "AlwaysTRUE" AND "Digitais"."MB-04-YSH";
   IF #_w4 THEN "MB_04_VEL" := REAL_TO_INT("PID".AUX_CALC[4]); END_IF;
   IF #_w4 AND "COMANDOS"."MB-04-HS1" THEN
       "PID".AUX_CALC[4] := "PID"."VA-PID-EEEB" * "PID".AUX_CALC[5];
   END_IF;
   IF #_w4 AND NOT "COMANDOS"."MB-04-HS1" THEN
       "PID".AUX_CALC[4] := "SETPOINTS"."MB-04-SP" * "PID".AUX_CALC[5];
   END_IF;
END_REGION
END_ORGANIZATION_BLOCK

FUNCTION_BLOCK "DANFOSS_REV"   // FB206, LAD
TITLE = CONTROLE INVERSOR SINAMICS
{ S7_Optimized_Access := 'FALSE' }
VERSION : 0.1
// stored: AutoNumber false, IsIECCheckEnabled false, SetENOAutomatically false, UDAEnableTagReadback false
   VAR_INPUT
      DBNO : Int;   // Número do DB
      DBPOS : Int;   // Posição do DB
      MF1 : Bool;   // Motor em falha
      MF2 : Bool;   // Motor em falha
      HM : Bool;   // Habilita manual
      HA : Bool;   // Habilita automático
      HAR : Bool;   // Habilita automático reverso
      CMA : Bool;   // Comando liga automático
      CLM : Bool;   // Comando liga manual
      CLMR : Bool;   // Comando liga manual reverso
      CDM : Bool;   // Comando desliga manual
      CRF : Bool;   // Comando reset de falha
      CRTO : Bool;   // Comando reset tepo de operação
      CHC : Bool;   // Comando habilita controle de velocidade
      CHB : Bool;   // Comando habilita bloqueio
      CL1S : Bool;   // Pulso a cada 1 segundo
      SRC : Bool;   // Status rede de comunicação
      FMM : Real;   // Fundo de escala frequência do motor
      SPM : Real;   // Setpoint manual de velocidade
      SPA : Real;   // Setpoint automático de velocidade
   END_VAR
   VAR_OUTPUT
      YFL : Bool;   // Indicação de falha no inversor
      YFPP : Bool;   // Indicação de falha no acionamento
      YR : Bool;   // Indicação de chave na posição remota
      YSH : Bool;   // Indicação de motor ligado
      YF : Bool;   // Indicação de motor em falha
      CL : Bool;   // Comando liga motor
      REV : Bool;   // Indicação de motor ligado no sentido reverso
      CMD_RESET : Bool;   // Reset de falha
      IN18 : Bool;   // ENTRADA DIGITAL
      IN19 : Bool;   // ENTRADA DIGITAL
      IN27 : Bool;   // ENTRADA DIGITAL
      IN29 : Bool;   // ENTRADA DIGITAL
      IN32 : Bool;   // ENTRADA DIGITAL
      IN33 : Bool;   // ENTRADA DIGITAL
      IT : Real;   // Indicação de corrente
      ST : Real;   // Indicação de frequência
   END_VAR
   VAR_IN_OUT
      SEG : Int;   // Segundos de operação
      MIN : Int;   // Minutos de operação
      HOR : Int;   // Horas de operação
   END_VAR
   VAR DB_SPECIFIC
      STW { ExternalAccessible := 'False'; ExternalVisible := 'False'; ExternalWritable := 'False'} : Struct   // PALAVRA DE STATUS DO INVERSOR
         SpeddRef { ExternalAccessible := 'False'; ExternalVisible := 'False'; ExternalWritable := 'False'} : Bool;   // Velocidade=Setpoint
         BUS { ExternalAccessible := 'False'; ExternalVisible := 'False'; ExternalWritable := 'False'} : Bool;   // Controle pelo BUS
         FreqOK { ExternalAccessible := 'False'; ExternalVisible := 'False'; ExternalWritable := 'False'} : Bool;   // Frequecia OK
         Operation { ExternalAccessible := 'False'; ExternalVisible := 'False'; ExternalWritable := 'False'} : Bool;   // Em operação
         Drive { ExternalAccessible := 'False'; ExternalVisible := 'False'; ExternalWritable := 'False'} : Bool;   // Drive OK
         Voltage { ExternalAccessible := 'False'; ExternalVisible := 'False'; ExternalWritable := 'False'} : Bool;   // Tensão excedida
         Torque { ExternalAccessible := 'False'; ExternalVisible := 'False'; ExternalWritable := 'False'} : Bool;   // Torque excedido
         Thermal { ExternalAccessible := 'False'; ExternalVisible := 'False'; ExternalWritable := 'False'} : Bool;   // Térmico excedido
         Ready_forswitch_on { ExternalAccessible := 'False'; ExternalVisible := 'False'; ExternalWritable := 'False'} : Bool;   // Controle habilitado
         Ready { ExternalAccessible := 'False'; ExternalVisible := 'False'; ExternalWritable := 'False'} : Bool;   // Inversor pronto
         Running { ExternalAccessible := 'False'; ExternalVisible := 'False'; ExternalWritable := 'False'} : Bool;   // Em funcionamento
         Fault { ExternalAccessible := 'False'; ExternalVisible := 'False'; ExternalWritable := 'False'} : Bool;   // Falha ativa
         Error { ExternalAccessible := 'False'; ExternalVisible := 'False'; ExternalWritable := 'False'} : Bool;   // Erro ativo
         Reservado { ExternalAccessible := 'False'; ExternalVisible := 'False'; ExternalWritable := 'False'} : Bool;   // Reservado
         TripLock { ExternalAccessible := 'False'; ExternalVisible := 'False'; ExternalWritable := 'False'} : Bool;   // Inibição ativa
         Warning { ExternalAccessible := 'False'; ExternalVisible := 'False'; ExternalWritable := 'False'} : Bool;   // Advertência
      END_STRUCT;
      LPZD2 : Int;   // Velocidade do motor
      LPZD3 : Int;   // Corrente do motor
      LPZD4 : Struct   // Entradas digitais
         INX2 : Bool;   // Reservado
         INX3 : Bool;   // Reservado
         INX4 : Bool;   // Reservado
         INX5 : Bool;   // Reservado
         INX6 : Bool;   // Reservado
         INX7 : Bool;   // Reservado
         INX8 : Bool;   // Reservado
         INX9 : Bool;   // Reservado
         IN33 : Bool;   // Entrada terminal 33
         IN32 : Bool;   // Entrada terminal 32
         IN29 : Bool;   // Entrada terminal 29
         IN27 : Bool;   // Entrada terminal 27
         IN19 : Bool;   // Entrada terminal 19
         IN18 : Bool;   // Entrada terminal 18
         INX0 : Bool;   // Reservado
         INX1 : Bool;   // Reservado
      END_STRUCT;
      CTW { ExternalAccessible := 'False'; ExternalVisible := 'False'; ExternalWritable := 'False'} : Struct   // PALAVRA DE CONTROLE DO INVERSOR
         Jog { ExternalAccessible := 'False'; ExternalVisible := 'False'; ExternalWritable := 'False'} : Bool;   // Habilita jog
         RampSEL { ExternalAccessible := 'False'; ExternalVisible := 'False'; ExternalWritable := 'False'} : Bool;   // Seleção RAMPA1/2
         Control_plc { ExternalAccessible := 'False'; ExternalVisible := 'False'; ExternalWritable := 'False'} : Bool;   // Valida dados do PLC
         Relay1 { ExternalAccessible := 'False'; ExternalVisible := 'False'; ExternalWritable := 'False'} : Bool;   // Habilita partida sentido reverso
         Relay4 { ExternalAccessible := 'False'; ExternalVisible := 'False'; ExternalWritable := 'False'} : Bool;   // Controlador de velocidade habilitado
         Setup0 { ExternalAccessible := 'False'; ExternalVisible := 'False'; ExternalWritable := 'False'} : Bool;   // Seleção de setup bit0
         Setup1 { ExternalAccessible := 'False'; ExternalVisible := 'False'; ExternalWritable := 'False'} : Bool;   // Seleção de setup bit1
         Start_reverse { ExternalAccessible := 'False'; ExternalVisible := 'False'; ExternalWritable := 'False'} : Bool;   // Habilita partida sentido reverso
         LSB { ExternalAccessible := 'False'; ExternalVisible := 'False'; ExternalWritable := 'False'} : Bool;   // Seleção externa LSB
         MSB { ExternalAccessible := 'False'; ExternalVisible := 'False'; ExternalWritable := 'False'} : Bool;   // Seleção externa MSB
         DCbrakeRamp { ExternalAccessible := 'False'; ExternalVisible := 'False'; ExternalWritable := 'False'} : Bool;   // Freio DC/Rampa
         Coasting { ExternalAccessible := 'False'; ExternalVisible := 'False'; ExternalWritable := 'False'} : Bool;   // Liga motor
         Enable_Ramp { ExternalAccessible := 'False'; ExternalVisible := 'False'; ExternalWritable := 'False'} : Bool;   // Habilita rampa
         Enable_ramp_generator { ExternalAccessible := 'False'; ExternalVisible := 'False'; ExternalWritable := 'False'} : Bool;   // Habilita gerador de rampa
         Start { ExternalAccessible := 'False'; ExternalVisible := 'False'; ExternalWritable := 'False'} : Bool;   // Liga motor
         Reset { ExternalAccessible := 'False'; ExternalVisible := 'False'; ExternalWritable := 'False'} : Bool;   // Reconhecimento de falha
      END_STRUCT;
      CT_MotorReference : Int;   // Referência de velocidade
      EPZD3 : Int;   // Reserva
      EPZD4 : Int;   // Reserva
      RESET : Bool;   // Reset de falha
      AUX01 : Bool;   // Auxiliar utilizado na lógica
      AUX02 : Bool;   // Auxiliar utilizado na lógica
      AUX03 : Bool;   // Auxiliar utilizado na lógica
      AUX04 : Bool;   // Auxiliar utilizado na lógica
      AUX05 : Bool;   // Auxiliar utilizado na lógica
      AUX06 : Bool;   // Auxiliar utilizado na lógica
      AUX07 : Bool;   // Auxiliar utilizado na lógica
      AUX08 : Bool;   // Auxiliar utilizado na lógica
      AUX09 : Bool;   // Auxiliar utilizado na lógica
      AUX10 : Bool;   // Auxiliar utilizado na lógica
      P60S : Bool;   // Pulso de 60 segundos
      P60M : Bool;   // Pulso de 60 minutos
      PFHO : Bool;   // Pulso de limite de horas
      SPS : Real;   // Frequência para controle
      TPP1 { S7_SetPoint := 'True'} : TON_TIME;   // Temporizador falha no acionamento
      TPP2 { S7_SetPoint := 'True'} : TON_TIME;   // Temporizador falha no acionamento
      TR { S7_SetPoint := 'True'} : TON_TIME;   // Temporizador reset de falha
   END_VAR
   VAR_TEMP
      LIGADO : Bool;   // Ligado
      FALHA : Bool;   // Falha
      TEMP0 : Bool;
      TEMP1 : Bool;
      ET_TPP1 : Time;   // Efetivo temporizador
      ET_TPP2 : Time;   // Efetivo temporizador
      ET_TR : Time;   // Efetivo temporizador
      AUXDB : Int;   // Auxiliar movimentação do DB
      ST1 : Real;   // Frequência convertida
   END_VAR
   VAR_TEMP   // added for the SCL form of the ladder/FBD networks
      _w1 : Bool;
      _w2 : Bool;
      _w3 : Bool;
      _w4 : Bool;
   END_VAR
BEGIN

NETWORK
TITLE = Leitura de dados da rede
//CARREGA O ENDEREÇO DA PRIMEIRA WORD DE ENTRADA

      L     #DBNO;  // Carrega n° da DB
      T     #AUXDB;

      OPN   DB [#AUXDB];  // Abre DB

      L     #DBPOS;  // Multiplica valor da posição para acertar ponteiro (valor x 8bit´s)
      L     8;
      *I;
      LAR1;  // Carrega valor de ponteiro no registrador 1

      L     DBW [AR1, P#0.0];
      T     %DIW34;
      L     DBW [AR1, P#2.0];
      T     #LPZD2;
      L     DBW [AR1, P#4.0];
      T     #LPZD3;
      L     DBW [AR1, P#6.0];
      T     %DIW40;

NETWORK
TITLE = CONVERSÃO DA LEITURA DE FREQUÊNCIA/CORRENTE
      L     #LPZD2;
      ITD;
      DTR;
      L     #FMM;
      *R;
      L     16384.0;
      /R;
      T     #ST;

      L     #LPZD3;
      ITD;
      DTR;
      L     100.0;
      /R;
      T     #IT;

NETWORK
TITLE = STATUS DO INVERSOR
// VERIFICA ESTADO DO PRIMEIRO BYTE DA PALAVRA DE ENTRADA  (PZD)

      A     #STW.Fault;
      =     #YFL;  //ALARME DE FALHA NO INVERSOR

// LEITURA DAS ENTRADAS DIGITAIS

      A     #LPZD4.IN33;  // ENTRADA DIGITAL DE REMOTO
      A     #STW.BUS;
      =     #YR;
      =     #IN33;

      A     #LPZD4.IN18;  // TERMINAL 18
      =     #IN18;

      A     #LPZD4.IN19;  // TERMINAL 19
      =     #IN19;

      A     #LPZD4.IN27;  // TERMINAL 27
      =     #IN27;

      A     #LPZD4.IN32;  // TERMINAL 32
      =     #IN32;

      A     #LPZD4.IN29;  // TERMINAL 29
      =     #IN29;

REGION Network 4: STATUS DE LIGADO
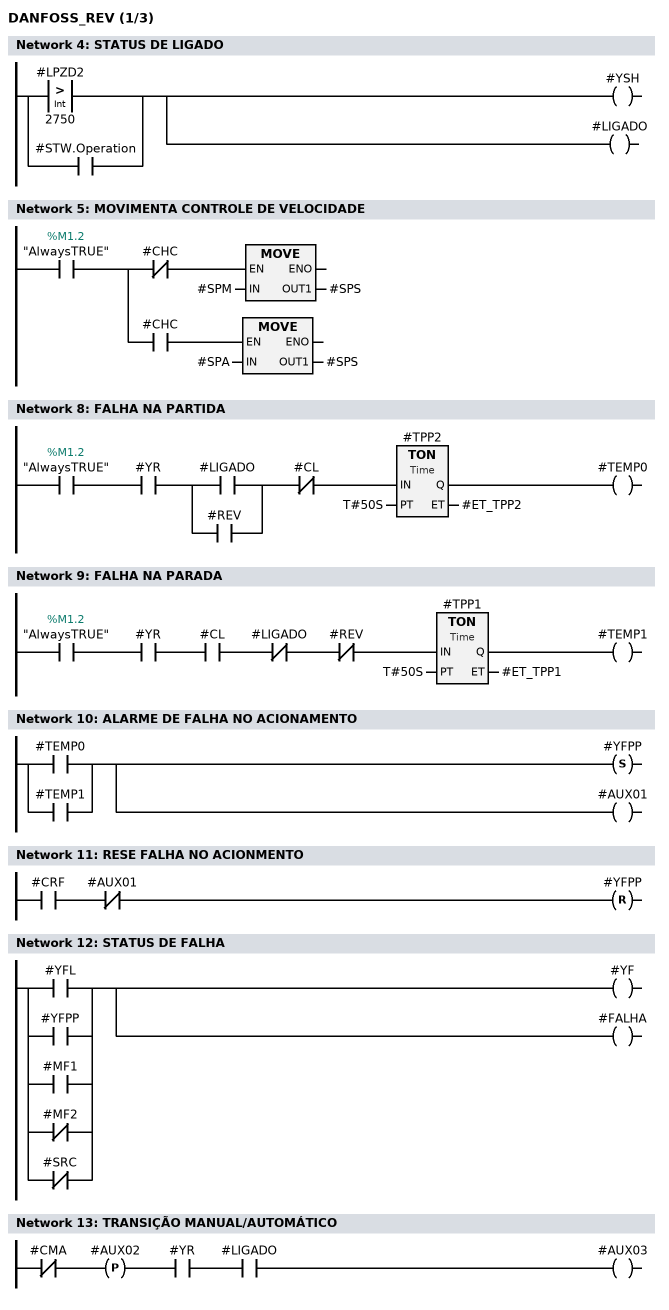
   RUNG wire#powerrail
      { S7_Templates := "SrcType := Int" } GT_Contact(in1 := #LPZD2, in2 := 2750)
      wire#w1
      Coil( #YSH )
   END_RUNG
   RUNG wire#powerrail
      Contact( #STW.Operation )
   END_RUNG wire#w1
   RUNG wire#w1
      Coil( #LIGADO )
   END_RUNG
   // the same network as SCL:
   #YSH := (#LPZD2 > 2750) OR #STW.Operation;
   #LIGADO := #YSH;
END_REGION

REGION Network 5: MOVIMENTA CONTROLE DE VELOCIDADE
   RUNG wire#powerrail
      Contact( "AlwaysTRUE" )
      wire#w1
      I_Contact( #CHC )
      { S7_GenerateENO := "TRUE" } Move(in := #SPM, out1 => #SPS)
   END_RUNG
   RUNG wire#w1
      Contact( #CHC )
      { S7_GenerateENO := "TRUE" } Move(in := #SPA, out1 => #SPS)
   END_RUNG
   // the same network as SCL:
   IF "AlwaysTRUE" AND NOT #CHC THEN #SPS := #SPM; END_IF;
   IF "AlwaysTRUE" AND #CHC THEN #SPS := #SPA; END_IF;
END_REGION

NETWORK
TITLE = Escreve setpoint de velocidade no inversor
      L     16384.0;  //Divide para encontrar a relação de conversão
      L     #SPS;
      *R;

      L     #FMM;  //Multiplica setpoint por fator para envio ao inversor
      /R;
      RND;
      T     #CT_MotorReference;


NETWORK
TITLE = ESCRITA DE DADOS NO INVERSOR
      +AR1  P#20.0;  //Carrega posição de escrita da DB

      L     %DIW42;
      T     DBW [AR1, P#0.0];  //Offset inicial
      L     #CT_MotorReference;
      T     DBW [AR1, P#2.0];


REGION Network 8: FALHA NA PARTIDA
   RUNG wire#powerrail
      Contact( "AlwaysTRUE" )
      Contact( #YR )
      wire#w1
      Contact( #LIGADO )
      wire#w2
      I_Contact( #CL )
      { S7_Templates := "time_type := Time" } #TPP2.TON(pt := T#50S, et => #ET_TPP2)
      Coil( #TEMP0 )
   END_RUNG
   RUNG wire#w1
      Contact( #REV )
   END_RUNG wire#w2
   // the same network as SCL:
   #TPP2(IN := "AlwaysTRUE" AND #YR AND (#LIGADO OR #REV) AND NOT #CL, PT := T#50S, ET => #ET_TPP2);   // TON
   #TEMP0 := #TPP2.Q;
END_REGION

REGION Network 9: FALHA NA PARADA
   RUNG wire#powerrail
      Contact( "AlwaysTRUE" )
      Contact( #YR )
      Contact( #CL )
      I_Contact( #LIGADO )
      I_Contact( #REV )
      { S7_Templates := "time_type := Time" } #TPP1.TON(pt := T#50S, et => #ET_TPP1)
      Coil( #TEMP1 )
   END_RUNG
   // the same network as SCL:
   #TPP1(IN := "AlwaysTRUE" AND #YR AND #CL AND NOT #LIGADO AND NOT #REV, PT := T#50S, ET => #ET_TPP1);   // TON
   #TEMP1 := #TPP1.Q;
END_REGION

REGION Network 10: ALARME DE FALHA NO ACIONAMENTO
   RUNG wire#powerrail
      Contact( #TEMP0 )
      wire#w1
      S_Coil( #YFPP )
   END_RUNG
   RUNG wire#powerrail
      Contact( #TEMP1 )
   END_RUNG wire#w1
   RUNG wire#w1
      Coil( #AUX01 )
   END_RUNG
   // the same network as SCL:
   #_w1 := #TEMP0 OR #TEMP1;
   IF #_w1 THEN #YFPP := TRUE; END_IF;
   #AUX01 := #_w1;
END_REGION

REGION Network 11: RESE FALHA NO ACIONMENTO
   RUNG wire#powerrail
      Contact( #CRF )
      I_Contact( #AUX01 )
      R_Coil( #YFPP )
   END_RUNG
   // the same network as SCL:
   IF #CRF AND NOT #AUX01 THEN #YFPP := FALSE; END_IF;
END_REGION

REGION Network 12: STATUS DE FALHA
   RUNG wire#powerrail
      Contact( #YFL )
      wire#w1
      Coil( #YF )
   END_RUNG
   RUNG wire#powerrail
      Contact( #YFPP )
   END_RUNG wire#w1
   RUNG wire#powerrail
      Contact( #MF1 )
   END_RUNG wire#w1
   RUNG wire#powerrail
      I_Contact( #MF2 )
   END_RUNG wire#w1
   RUNG wire#powerrail
      I_Contact( #SRC )
   END_RUNG wire#w1
   RUNG wire#w1
      Coil( #FALHA )
   END_RUNG
   // the same network as SCL:
   #YF := #YFL OR #YFPP OR #MF1 OR NOT #MF2 OR NOT #SRC;
   #FALHA := #YF;
END_REGION

REGION Network 13: TRANSIÇÃO MANUAL/AUTOMÁTICO
   RUNG wire#powerrail
      I_Contact( #CMA )
      P_Trig( #AUX02 )
      Contact( #YR )
      Contact( #LIGADO )
      Coil( #AUX03 )
   END_RUNG
   // the same network as SCL:
   #_w1 := NOT #CMA AND NOT #AUX02;   // rising edge
   #AUX02 := NOT #CMA;
   #AUX03 := #_w1 AND #YR AND #LIGADO;
END_REGION

REGION Network 14: COMANDO LIGA MANUAL SENTIDO DIRETO
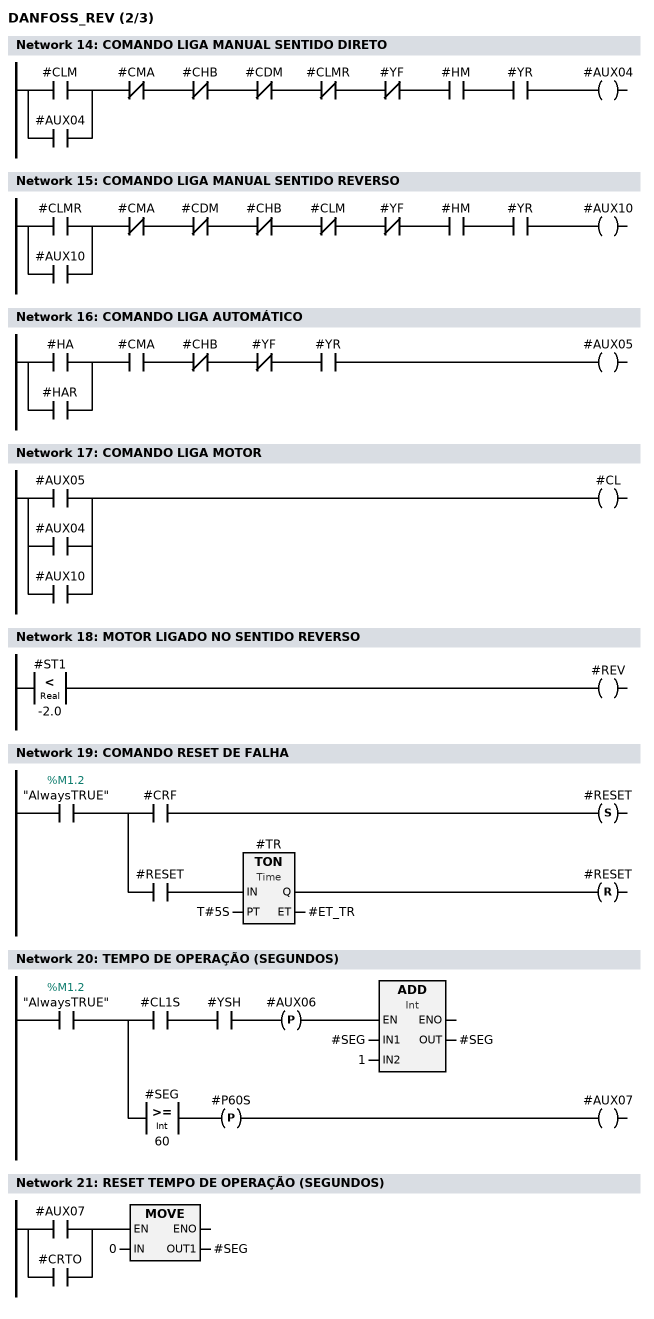
   RUNG wire#powerrail
      Contact( #CLM )
      wire#w1
      I_Contact( #CMA )
      I_Contact( #CHB )
      I_Contact( #CDM )
      I_Contact( #CLMR )
      I_Contact( #YF )
      Contact( #HM )
      Contact( #YR )
      Coil( #AUX04 )
   END_RUNG
   RUNG wire#powerrail
      Contact( #AUX04 )
   END_RUNG wire#w1
   // the same network as SCL:
   #AUX04 := (#CLM OR #AUX04) AND NOT #CMA AND NOT #CHB AND NOT #CDM AND NOT #CLMR AND NOT #YF AND #HM AND #YR;
END_REGION

REGION Network 15: COMANDO LIGA MANUAL SENTIDO REVERSO
   RUNG wire#powerrail
      Contact( #CLMR )
      wire#w1
      I_Contact( #CMA )
      I_Contact( #CDM )
      I_Contact( #CHB )
      I_Contact( #CLM )
      I_Contact( #YF )
      Contact( #HM )
      Contact( #YR )
      Coil( #AUX10 )
   END_RUNG
   RUNG wire#powerrail
      Contact( #AUX10 )
   END_RUNG wire#w1
   // the same network as SCL:
   #AUX10 := (#CLMR OR #AUX10) AND NOT #CMA AND NOT #CDM AND NOT #CHB AND NOT #CLM AND NOT #YF AND #HM AND #YR;
END_REGION

REGION Network 16: COMANDO LIGA AUTOMÁTICO
   RUNG wire#powerrail
      Contact( #HA )
      wire#w1
      Contact( #CMA )
      I_Contact( #CHB )
      I_Contact( #YF )
      Contact( #YR )
      Coil( #AUX05 )
   END_RUNG
   RUNG wire#powerrail
      Contact( #HAR )
   END_RUNG wire#w1
   // the same network as SCL:
   #AUX05 := (#HA OR #HAR) AND #CMA AND NOT #CHB AND NOT #YF AND #YR;
END_REGION

REGION Network 17: COMANDO LIGA MOTOR
   RUNG wire#powerrail
      Contact( #AUX05 )
      wire#w1
      Coil( #CL )
   END_RUNG
   RUNG wire#powerrail
      Contact( #AUX04 )
   END_RUNG wire#w1
   RUNG wire#powerrail
      Contact( #AUX10 )
   END_RUNG wire#w1
   // the same network as SCL:
   #CL := #AUX05 OR #AUX04 OR #AUX10;
END_REGION

REGION Network 18: MOTOR LIGADO NO SENTIDO REVERSO
   RUNG wire#powerrail
      { S7_Templates := "SrcType := Real" } LT_Contact(in1 := #ST1, in2 := -2.0)
      Coil( #REV )
   END_RUNG
   // the same network as SCL:
   #REV := #ST1 < (-2.0);
END_REGION

REGION Network 19: COMANDO RESET DE FALHA
   RUNG wire#powerrail
      Contact( "AlwaysTRUE" )
      wire#w1
      Contact( #CRF )
      S_Coil( #RESET )
   END_RUNG
   RUNG wire#w1
      Contact( #RESET )
      { S7_Templates := "time_type := Time" } #TR.TON(pt := T#5S, et => #ET_TR)
      R_Coil( #RESET )
   END_RUNG
   // the same network as SCL:
   IF "AlwaysTRUE" AND #CRF THEN #RESET := TRUE; END_IF;
   #TR(IN := "AlwaysTRUE" AND #RESET, PT := T#5S, ET => #ET_TR);   // TON
   IF #TR.Q THEN #RESET := FALSE; END_IF;
END_REGION

REGION Network 20: TEMPO DE OPERAÇÃO (SEGUNDOS)
   RUNG wire#powerrail
      Contact( "AlwaysTRUE" )
      wire#w1
      Contact( #CL1S )
      Contact( #YSH )
      P_Trig( #AUX06 )
      { S7_Templates := "SrcType := Int"; S7_GenerateENO := "TRUE" } Add(in1 := #SEG, in2 := 1, out => #SEG)
   END_RUNG
   RUNG wire#w1
      { S7_Templates := "SrcType := Int" } GE_Contact(in1 := #SEG, in2 := 60)
      P_Trig( #P60S )
      Coil( #AUX07 )
   END_RUNG
   // the same network as SCL:
   #_w1 := "AlwaysTRUE" AND #CL1S AND #YSH;
   #_w2 := #_w1 AND NOT #AUX06;   // rising edge
   #AUX06 := #_w1;
   IF #_w2 THEN #SEG := #SEG + 1; END_IF;
   #_w3 := "AlwaysTRUE" AND (#SEG >= 60);
   #_w4 := #_w3 AND NOT #P60S;   // rising edge
   #P60S := #_w3;
   #AUX07 := #_w4;
END_REGION

REGION Network 21: RESET TEMPO DE OPERAÇÃO (SEGUNDOS)
   RUNG wire#powerrail
      Contact( #AUX07 )
      wire#w1
      { S7_GenerateENO := "TRUE" } Move(in := 0, out1 => #SEG)
   END_RUNG
   RUNG wire#powerrail
      Contact( #CRTO )
   END_RUNG wire#w1
   // the same network as SCL:
   IF #AUX07 OR #CRTO THEN #SEG := 0; END_IF;
END_REGION

REGION Network 22: TEMPO DE OPERAÇÃO (MINUTOS)
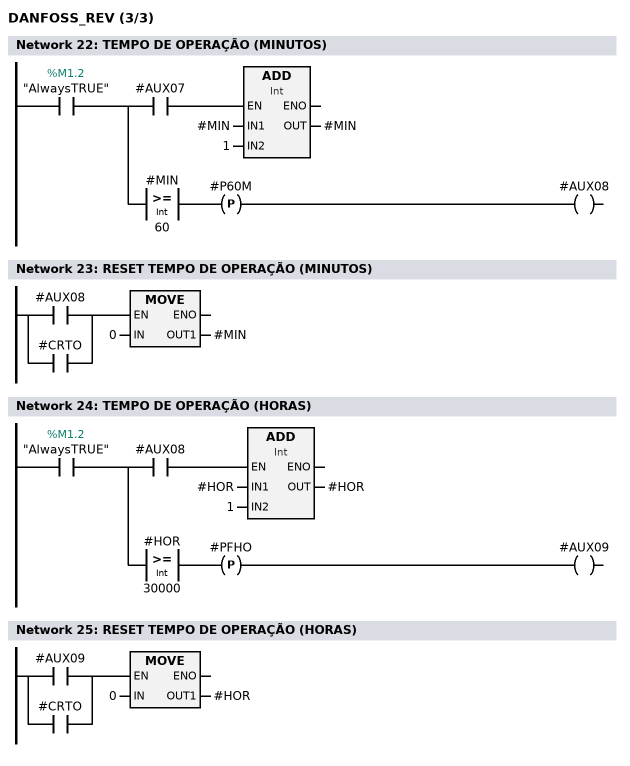
   RUNG wire#powerrail
      Contact( "AlwaysTRUE" )
      wire#w1
      Contact( #AUX07 )
      { S7_Templates := "SrcType := Int"; S7_GenerateENO := "TRUE" } Add(in1 := #MIN, in2 := 1, out => #MIN)
   END_RUNG
   RUNG wire#w1
      { S7_Templates := "SrcType := Int" } GE_Contact(in1 := #MIN, in2 := 60)
      P_Trig( #P60M )
      Coil( #AUX08 )
   END_RUNG
   // the same network as SCL:
   IF "AlwaysTRUE" AND #AUX07 THEN #MIN := #MIN + 1; END_IF;
   #_w1 := "AlwaysTRUE" AND (#MIN >= 60);
   #_w2 := #_w1 AND NOT #P60M;   // rising edge
   #P60M := #_w1;
   #AUX08 := #_w2;
END_REGION

REGION Network 23: RESET TEMPO DE OPERAÇÃO (MINUTOS)
   RUNG wire#powerrail
      Contact( #AUX08 )
      wire#w1
      { S7_GenerateENO := "TRUE" } Move(in := 0, out1 => #MIN)
   END_RUNG
   RUNG wire#powerrail
      Contact( #CRTO )
   END_RUNG wire#w1
   // the same network as SCL:
   IF #AUX08 OR #CRTO THEN #MIN := 0; END_IF;
END_REGION

REGION Network 24: TEMPO DE OPERAÇÃO (HORAS)
   RUNG wire#powerrail
      Contact( "AlwaysTRUE" )
      wire#w1
      Contact( #AUX08 )
      { S7_Templates := "SrcType := Int"; S7_GenerateENO := "TRUE" } Add(in1 := #HOR, in2 := 1, out => #HOR)
   END_RUNG
   RUNG wire#w1
      { S7_Templates := "SrcType := Int" } GE_Contact(in1 := #HOR, in2 := 30000)
      P_Trig( #PFHO )
      Coil( #AUX09 )
   END_RUNG
   // the same network as SCL:
   IF "AlwaysTRUE" AND #AUX08 THEN #HOR := #HOR + 1; END_IF;
   #_w1 := "AlwaysTRUE" AND (#HOR >= 30000);
   #_w2 := #_w1 AND NOT #PFHO;   // rising edge
   #PFHO := #_w1;
   #AUX09 := #_w2;
END_REGION

REGION Network 25: RESET TEMPO DE OPERAÇÃO (HORAS)
   RUNG wire#powerrail
      Contact( #AUX09 )
      wire#w1
      { S7_GenerateENO := "TRUE" } Move(in := 0, out1 => #HOR)
   END_RUNG
   RUNG wire#powerrail
      Contact( #CRTO )
   END_RUNG wire#w1
   // the same network as SCL:
   IF #AUX09 OR #CRTO THEN #HOR := 0; END_IF;
END_REGION

NETWORK
TITLE = ESCRITA DOS DADOS NO INVERSOR (PALAVRA DE COMANDO)
      A     "AlwaysTRUE";
      =     #CTW.DCbrakeRamp;
      =     #CTW.Coasting;
      =     #CTW.Enable_Ramp;
      =     #CTW.Enable_ramp_generator;
      =     #CTW.Control_plc;  //Valida setpoint


      A     #CL;
      =     #CTW.Start;  //LIGA/DESL

      A     #CL;
      A     #AUX10;
      A     #HAR;
      =     #CTW.Start_reverse;  //LIGA/DESL REVERSO


      A     #RESET;
      AN    #CL;
      =     #CTW.Reset;  //RESET
END_FUNCTION_BLOCK

